   1:  PR[91,1] = PR[90,1] + -34.385;
   1:  PR[91,2] = PR[90,2] + -12.687;
   1:L PR[91] R[100]mm/sec CNT100;
   1:  PR[91,1] = PR[90,1] + -33.183;
   1:  PR[91,2] = PR[90,2] + -13.979;
   1:L PR[91] R[100]mm/sec CNT100;
   1:  PR[91,1] = PR[90,1] + -31.805;
   1:  PR[91,2] = PR[90,2] + -15.148;
   1:L PR[91] R[100]mm/sec CNT100;
   1:  PR[91,1] = PR[90,1] + -30.132;
   1:  PR[91,2] = PR[90,2] + -16.456;
   1:L PR[91] R[100]mm/sec CNT100;
   1:  PR[91,1] = PR[90,1] + -27.677;
   1:  PR[91,2] = PR[90,2] + -17.817;
   1:L PR[91] R[100]mm/sec CNT100;
   1:  PR[91,1] = PR[90,1] + -27.017;
   1:  PR[91,2] = PR[90,2] + -18.151;
   1:L PR[91] R[100]mm/sec CNT100;
   1:  PR[91,1] = PR[90,1] + -24.103;
   1:  PR[91,2] = PR[90,2] + -19.209;
   1:L PR[91] R[100]mm/sec CNT100;
   1:  PR[91,1] = PR[90,1] + -20.848;
   1:  PR[91,2] = PR[90,2] + -19.885;
   1:L PR[91] R[100]mm/sec CNT100;
   1:  PR[91,1] = PR[90,1] + -20.625;
   1:  PR[91,2] = PR[90,2] + -19.911;
   1:L PR[91] R[100]mm/sec CNT100;
   1:  PR[91,1] = PR[90,1] + -17.368;
   1:  PR[91,2] = PR[90,2] + -20.082;
   1:L PR[91] R[100]mm/sec CNT100;
   1:  PR[91,1] = PR[90,1] + -14.474;
   1:  PR[91,2] = PR[90,2] + -19.791;
   1:L PR[91] R[100]mm/sec CNT100;
   1:  PR[91,1] = PR[90,1] + -13.607;
   1:  PR[91,2] = PR[90,2] + -19.670;
   1:L PR[91] R[100]mm/sec CNT100;
   1:  PR[91,1] = PR[90,1] + -10.936;
   1:  PR[91,2] = PR[90,2] + -18.979;
   1:L PR[91] R[100]mm/sec CNT100;
   1:  PR[91,1] = PR[90,1] + -8.588;
   1:  PR[91,2] = PR[90,2] + -17.949;
   1:L PR[91] R[100]mm/sec CNT100;
   1:  PR[91,1] = PR[90,1] + -7.248;
   1:  PR[91,2] = PR[90,2] + -17.378;
   1:L PR[91] R[100]mm/sec CNT100;
   1:  PR[91,1] = PR[90,1] + -5.237;
   1:  PR[91,2] = PR[90,2] + -16.092;
   1:L PR[91] R[100]mm/sec CNT100;
   1:  PR[91,1] = PR[90,1] + -4.843;
   1:  PR[91,2] = PR[90,2] + -15.808;
   1:L PR[91] R[100]mm/sec CNT100;
   1:  PR[91,1] = PR[90,1] + -2.769;
   1:  PR[91,2] = PR[90,2] + -13.975;
   1:L PR[91] R[100]mm/sec CNT100;
   1:  PR[91,1] = PR[90,1] + -2.120;
   1:  PR[91,2] = PR[90,2] + -13.214;
   1:L PR[91] R[100]mm/sec CNT100;
   1:  PR[91,1] = PR[90,1] + -1.676;
   1:  PR[91,2] = PR[90,2] + -12.857;
   1:L PR[91] R[100]mm/sec CNT100;
   1:  PR[91,1] = PR[90,1] + -0.501;
   1:  PR[91,2] = PR[90,2] + -12.027;
   1:L PR[91] R[100]mm/sec CNT100;
   1:  PR[91,1] = PR[90,1] + 0.440;
   1:  PR[91,2] = PR[90,2] + -12.361;
   1:L PR[91] R[100]mm/sec CNT100;
   1:  PR[91,1] = PR[90,1] + 1.193;
   1:L PR[91] R[100]mm/sec CNT100;
   1:  PR[91,1] = PR[90,1] + 1.817;
   1:  PR[91,2] = PR[90,2] + -12.872;
   1:L PR[91] R[100]mm/sec CNT100;
   1:  PR[91,1] = PR[90,1] + 2.256;
   1:  PR[91,2] = PR[90,2] + -13.184;
   1:L PR[91] R[100]mm/sec CNT100;
   1:  PR[91,1] = PR[90,1] + 2.936;
   1:  PR[91,2] = PR[90,2] + -13.984;
   1:L PR[91] R[100]mm/sec CNT100;
   1:  PR[91,1] = PR[90,1] + 4.982;
   1:  PR[91,2] = PR[90,2] + -15.795;
   1:L PR[91] R[100]mm/sec CNT100;
   1:  PR[91,1] = PR[90,1] + 6.799;
   1:  PR[91,2] = PR[90,2] + -16.959;
   1:L PR[91] R[100]mm/sec CNT100;
   1:  PR[91,1] = PR[90,1] + 7.427;
   1:  PR[91,2] = PR[90,2] + -17.391;
   1:L PR[91] R[100]mm/sec CNT100;
   1:  PR[91,1] = PR[90,1] + 11.082;
   1:  PR[91,2] = PR[90,2] + -18.974;
   1:L PR[91] R[100]mm/sec CNT100;
   1:  PR[91,1] = PR[90,1] + 13.736;
   1:  PR[91,2] = PR[90,2] + -19.662;
   1:L PR[91] R[100]mm/sec CNT100;
   1:  PR[91,1] = PR[90,1] + 16.945;
   1:  PR[91,2] = PR[90,2] + -19.998;
   1:L PR[91] R[100]mm/sec CNT100;
   1:  PR[91,1] = PR[90,1] + 17.542;
   1:  PR[91,2] = PR[90,2] + -20.081;
   1:L PR[91] R[100]mm/sec CNT100;
   1:  PR[91,1] = PR[90,1] + 20.757;
   1:  PR[91,2] = PR[90,2] + -19.914;
   1:L PR[91] R[100]mm/sec CNT100;
   1:  PR[91,1] = PR[90,1] + 20.981;
   1:  PR[91,2] = PR[90,2] + -19.888;
   1:L PR[91] R[100]mm/sec CNT100;
   1:  PR[91,1] = PR[90,1] + 24.231;
   1:  PR[91,2] = PR[90,2] + -19.216;
   1:L PR[91] R[100]mm/sec CNT100;
   1:  PR[91,1] = PR[90,1] + 27.158;
   1:  PR[91,2] = PR[90,2] + -18.158;
   1:L PR[91] R[100]mm/sec CNT100;
   1:  PR[91,1] = PR[90,1] + 27.815;
   1:  PR[91,2] = PR[90,2] + -17.826;
   1:L PR[91] R[100]mm/sec CNT100;
   1:  PR[91,1] = PR[90,1] + 30.243;
   1:  PR[91,2] = PR[90,2] + -16.487;
   1:L PR[91] R[100]mm/sec CNT100;
   1:  PR[91,1] = PR[90,1] + 31.424;
   1:  PR[91,2] = PR[90,2] + -15.490;
   1:L PR[91] R[100]mm/sec CNT100;
   1:  PR[91,1] = PR[90,1] + 33.327;
   1:  PR[91,2] = PR[90,2] + -13.989;
   1:L PR[91] R[100]mm/sec CNT100;
   1:  PR[91,1] = PR[90,1] + 34.543;
   1:  PR[91,2] = PR[90,2] + -12.683;
   1:L PR[91] R[100]mm/sec CNT100;
   1:  PR[91,1] = PR[90,1] + 35.930;
   1:  PR[91,2] = PR[90,2] + -10.746;
   1:L PR[91] R[100]mm/sec CNT100;
   1:  PR[91,1] = PR[90,1] + 36.829;
   1:  PR[91,2] = PR[90,2] + -9.386;
   1:L PR[91] R[100]mm/sec CNT100;
   1:  PR[91,1] = PR[90,1] + 37.404;
   1:  PR[91,2] = PR[90,2] + -8.113;
   1:L PR[91] R[100]mm/sec CNT100;
   1:  PR[91,1] = PR[90,1] + 38.431;
   1:  PR[91,2] = PR[90,2] + -5.567;
   1:L PR[91] R[100]mm/sec CNT100;
   1:  PR[91,1] = PR[90,1] + 38.718;
   1:  PR[91,2] = PR[90,2] + -4.469;
   1:L PR[91] R[100]mm/sec CNT100;
   1:  PR[91,1] = PR[90,1] + 39.102;
   1:  PR[91,2] = PR[90,2] + -1.437;
   1:L PR[91] R[100]mm/sec CNT100;
   1:  PR[91,1] = PR[90,1] + 39.190;
   1:  PR[91,2] = PR[90,2] + -0.345;
   1:L PR[91] R[100]mm/sec CNT100;
   1:  PR[91,1] = PR[90,1] + 38.810;
   1:  PR[91,2] = PR[90,2] + 2.635;
   1:L PR[91] R[100]mm/sec CNT100;
   1:  PR[91,1] = PR[90,1] + 38.710;
   1:  PR[91,2] = PR[90,2] + 3.878;
   1:L PR[91] R[100]mm/sec CNT100;
   1:  PR[91,1] = PR[90,1] + 38.430;
   1:  PR[91,2] = PR[90,2] + 4.944;
   1:L PR[91] R[100]mm/sec CNT100;
   1:  PR[91,1] = PR[90,1] + 37.403;
   1:  PR[91,2] = PR[90,2] + 7.490;
   1:L PR[91] R[100]mm/sec CNT100;
   1:  PR[91,1] = PR[90,1] + 36.840;
   1:  PR[91,2] = PR[90,2] + 8.736;
   1:L PR[91] R[100]mm/sec CNT100;
   1:  PR[91,1] = PR[90,1] + 35.420;
   1:  PR[91,2] = PR[90,2] + 10.708;
   1:L PR[91] R[100]mm/sec CNT100;
   1:  PR[91,1] = PR[90,1] + 34.521;
   1:  PR[91,2] = PR[90,2] + 12.083;
   1:L PR[91] R[100]mm/sec CNT100;
   1:  PR[91,1] = PR[90,1] + 33.307;
   1:  PR[91,2] = PR[90,2] + 13.386;
   1:L PR[91] R[100]mm/sec CNT100;
   1:  PR[91,1] = PR[90,1] + 31.932;
   1:  PR[91,2] = PR[90,2] + 14.555;
   1:L PR[91] R[100]mm/sec CNT100;
   1:  PR[91,1] = PR[90,1] + 30.267;
   1:  PR[91,2] = PR[90,2] + 15.850;
   1:L PR[91] R[100]mm/sec CNT100;
   1:  PR[91,1] = PR[90,1] + 27.814;
   1:  PR[91,2] = PR[90,2] + 17.202;
   1:L PR[91] R[100]mm/sec CNT100;
   1:  PR[91,1] = PR[90,1] + 27.157;
   1:  PR[91,2] = PR[90,2] + 17.534;
   1:L PR[91] R[100]mm/sec CNT100;
   1:  PR[91,1] = PR[90,1] + 24.231;
   1:  PR[91,2] = PR[90,2] + 18.592;
   1:L PR[91] R[100]mm/sec CNT100;
   1:  PR[91,1] = PR[90,1] + 20.982;
   1:  PR[91,2] = PR[90,2] + 19.264;
   1:L PR[91] R[100]mm/sec CNT100;
   1:  PR[91,1] = PR[90,1] + 20.758;
   1:  PR[91,2] = PR[90,2] + 19.290;
   1:L PR[91] R[100]mm/sec CNT100;
   1:  PR[91,1] = PR[90,1] + 17.520;
   1:  PR[91,2] = PR[90,2] + 19.459;
   1:L PR[91] R[100]mm/sec CNT100;
   1:  PR[91,1] = PR[90,1] + 14.634;
   1:  PR[91,2] = PR[90,2] + 19.166;
   1:L PR[91] R[100]mm/sec CNT100;
   1:  PR[91,1] = PR[90,1] + 13.768;
   1:  PR[91,2] = PR[90,2] + 19.046;
   1:L PR[91] R[100]mm/sec CNT100;
   1:  PR[91,1] = PR[90,1] + 11.095;
   1:  PR[91,2] = PR[90,2] + 18.353;
   1:L PR[91] R[100]mm/sec CNT100;
   1:  PR[91,1] = PR[90,1] + 8.749;
   1:  PR[91,2] = PR[90,2] + 17.327;
   1:L PR[91] R[100]mm/sec CNT100;
   1:  PR[91,1] = PR[90,1] + 7.438;
   1:  PR[91,2] = PR[90,2] + 16.779;
   1:L PR[91] R[100]mm/sec CNT100;
   1:  PR[91,1] = PR[90,1] + 5.424;
   1:  PR[91,2] = PR[90,2] + 15.493;
   1:L PR[91] R[100]mm/sec CNT100;
   1:  PR[91,1] = PR[90,1] + 5.171;
   1:  PR[91,2] = PR[90,2] + 15.318;
   1:L PR[91] R[100]mm/sec CNT100;
   1:  PR[91,1] = PR[90,1] + 4.692;
   1:  PR[91,2] = PR[90,2] + 14.939;
   1:L PR[91] R[100]mm/sec CNT100;
   1:  PR[91,1] = PR[90,1] + 3.034;
   1:  PR[91,2] = PR[90,2] + 13.458;
   1:L PR[91] R[100]mm/sec CNT100;
   1:  PR[91,1] = PR[90,1] + 2.330;
   1:  PR[91,2] = PR[90,2] + 12.730;
   1:L PR[91] R[100]mm/sec CNT100;
   1:  PR[91,1] = PR[90,1] + 2.090;
   1:  PR[91,2] = PR[90,2] + 12.413;
   1:L PR[91] R[100]mm/sec CNT100;
   1:  PR[91,1] = PR[90,1] + 1.443;
   1:  PR[91,2] = PR[90,2] + 11.955;
   1:L PR[91] R[100]mm/sec CNT100;
   1:  PR[91,1] = PR[90,1] + 0.740;
   1:  PR[91,2] = PR[90,2] + 11.570;
   1:L PR[91] R[100]mm/sec CNT100;
   1:  PR[91,1] = PR[90,1] + -0.586;
   1:L PR[91] R[100]mm/sec CNT100;
   1:  PR[91] = PR[90];
   1:  PR[91,1] = PR[90,1] + -1.541;
   1:  PR[91,2] = PR[90,2] + 12.321;
   1:  PR[91,3] = PR[90,3] + 28.365;
   1:L PR[91] R[100]mm/sec CNT100;
   1:  PR[91,1] = PR[90,1] + -1.870;
   1:  PR[91,2] = PR[90,2] + 12.749;
   1:L PR[91] R[100]mm/sec CNT100;
   1:  PR[91,1] = PR[90,1] + -2.109;
   1:  PR[91,2] = PR[90,2] + 12.974;
   1:L PR[91] R[100]mm/sec CNT100;
   1:  PR[91,1] = PR[90,1] + -2.678;
   1:  PR[91,2] = PR[90,2] + 13.569;
   1:L PR[91] R[100]mm/sec CNT100;
   1:  PR[91,1] = PR[90,1] + -4.236;
   1:  PR[91,2] = PR[90,2] + 14.958;
   1:L PR[91] R[100]mm/sec CNT100;
   1:  PR[91,1] = PR[90,1] + -4.761;
   1:  PR[91,2] = PR[90,2] + 15.373;
   1:L PR[91] R[100]mm/sec CNT100;
   1:  PR[91,1] = PR[90,1] + -6.588;
   1:  PR[91,2] = PR[90,2] + 16.543;
   1:L PR[91] R[100]mm/sec CNT100;
   1:  PR[91,1] = PR[90,1] + -7.022;
   1:  PR[91,2] = PR[90,2] + 16.834;
   1:L PR[91] R[100]mm/sec CNT100;
   1:  PR[91,1] = PR[90,1] + -9.377;
   1:  PR[91,2] = PR[90,2] + 17.863;
   1:L PR[91] R[100]mm/sec CNT100;
   1:  PR[91,1] = PR[90,1] + -10.739;
   1:  PR[91,2] = PR[90,2] + 18.434;
   1:L PR[91] R[100]mm/sec CNT100;
   1:  PR[91,1] = PR[90,1] + -13.266;
   1:  PR[91,2] = PR[90,2] + 19.087;
   1:L PR[91] R[100]mm/sec CNT100;
   1:  PR[91,1] = PR[90,1] + -16.330;
   1:  PR[91,2] = PR[90,2] + 19.406;
   1:L PR[91] R[100]mm/sec CNT100;
   1:  PR[91,1] = PR[90,1] + -17.174;
   1:  PR[91,2] = PR[90,2] + 19.521;
   1:L PR[91] R[100]mm/sec CNT100;
   1:  PR[91,1] = PR[90,1] + -20.260;
   1:  PR[91,2] = PR[90,2] + 19.358;
   1:L PR[91] R[100]mm/sec CNT100;
   1:  PR[91,1] = PR[90,1] + -20.724;
   1:  PR[91,2] = PR[90,2] + 19.304;
   1:L PR[91] R[100]mm/sec CNT100;
   1:  PR[91,1] = PR[90,1] + -23.832;
   1:  PR[91,2] = PR[90,2] + 18.659;
   1:L PR[91] R[100]mm/sec CNT100;
   1:  PR[91,1] = PR[90,1] + -26.964;
   1:  PR[91,2] = PR[90,2] + 17.504;
   1:L PR[91] R[100]mm/sec CNT100;
   1:  PR[91,1] = PR[90,1] + -29.926;
   1:  PR[91,2] = PR[90,2] + 15.872;
   1:L PR[91] R[100]mm/sec CNT100;
   1:  PR[91,1] = PR[90,1] + -30.643;
   1:  PR[91,2] = PR[90,2] + 15.268;
   1:L PR[91] R[100]mm/sec CNT100;
   1:  PR[91,1] = PR[90,1] + -32.892;
   1:  PR[91,2] = PR[90,2] + 13.488;
   1:L PR[91] R[100]mm/sec CNT100;
   1:  PR[91,1] = PR[90,1] + -34.331;
   1:  PR[91,2] = PR[90,2] + 11.939;
   1:L PR[91] R[100]mm/sec CNT100;
   1:  PR[91,1] = PR[90,1] + -35.417;
   1:  PR[91,2] = PR[90,2] + 10.423;
   1:L PR[91] R[100]mm/sec CNT100;
   1:  PR[91,1] = PR[90,1] + -36.499;
   1:  PR[91,2] = PR[90,2] + 8.777;
   1:L PR[91] R[100]mm/sec CNT100;
   1:  PR[91,1] = PR[90,1] + -37.206;
   1:  PR[91,2] = PR[90,2] + 7.190;
   1:L PR[91] R[100]mm/sec CNT100;
   1:  PR[91,1] = PR[90,1] + -38.062;
   1:  PR[91,2] = PR[90,2] + 5.058;
   1:L PR[91] R[100]mm/sec CNT100;
   1:  PR[91,1] = PR[90,1] + -38.428;
   1:  PR[91,2] = PR[90,2] + 3.643;
   1:L PR[91] R[100]mm/sec CNT100;
   1:  PR[91,1] = PR[90,1] + -38.751;
   1:  PR[91,2] = PR[90,2] + 1.099;
   1:L PR[91] R[100]mm/sec CNT100;
   1:  PR[91,1] = PR[90,1] + -38.860;
   1:  PR[91,2] = PR[90,2] + -0.277;
   1:L PR[91] R[100]mm/sec CNT100;
   1:  PR[91,1] = PR[90,1] + -38.538;
   1:  PR[91,2] = PR[90,2] + -2.788;
   1:L PR[91] R[100]mm/sec CNT100;
   1:  PR[91,1] = PR[90,1] + -38.420;
   1:  PR[91,2] = PR[90,2] + -4.301;
   1:L PR[91] R[100]mm/sec CNT100;
   1:  PR[91,1] = PR[90,1] + -38.062;
   1:  PR[91,2] = PR[90,2] + -5.682;
   1:L PR[91] R[100]mm/sec CNT100;
   1:  PR[91,1] = PR[90,1] + -37.206;
   1:  PR[91,2] = PR[90,2] + -7.814;
   1:L PR[91] R[100]mm/sec CNT100;
   1:  PR[91,1] = PR[90,1] + -36.512;
   1:  PR[91,2] = PR[90,2] + -9.372;
   1:L PR[91] R[100]mm/sec CNT100;
   1:  PR[91,1] = PR[90,1] + -35.356;
   1:  PR[91,2] = PR[90,2] + -10.976;
   1:L PR[91] R[100]mm/sec CNT100;
   1:  PR[91,1] = PR[90,1] + -34.309;
   1:  PR[91,2] = PR[90,2] + -12.587;
   1:L PR[91] R[100]mm/sec CNT100;
   1:  PR[91,1] = PR[90,1] + -32.875;
   1:  PR[91,2] = PR[90,2] + -14.130;
   1:L PR[91] R[100]mm/sec CNT100;
   1:  PR[91,1] = PR[90,1] + -31.875;
   1:  PR[91,2] = PR[90,2] + -14.979;
   1:L PR[91] R[100]mm/sec CNT100;
   1:  PR[91,1] = PR[90,1] + -29.950;
   1:  PR[91,2] = PR[90,2] + -16.483;
   1:L PR[91] R[100]mm/sec CNT100;
   1:  PR[91,1] = PR[90,1] + -26.964;
   1:  PR[91,2] = PR[90,2] + -18.128;
   1:L PR[91] R[100]mm/sec CNT100;
   1:  PR[91,1] = PR[90,1] + -23.830;
   1:  PR[91,2] = PR[90,2] + -19.283;
   1:L PR[91] R[100]mm/sec CNT100;
   1:  PR[91,1] = PR[90,1] + -20.722;
   1:  PR[91,2] = PR[90,2] + -19.928;
   1:L PR[91] R[100]mm/sec CNT100;
   1:  PR[91,1] = PR[90,1] + -20.256;
   1:  PR[91,2] = PR[90,2] + -19.982;
   1:L PR[91] R[100]mm/sec CNT100;
   1:  PR[91,1] = PR[90,1] + -17.142;
   1:  PR[91,2] = PR[90,2] + -20.146;
   1:L PR[91] R[100]mm/sec CNT100;
   1:  PR[91,1] = PR[90,1] + -14.376;
   1:  PR[91,2] = PR[90,2] + -19.868;
   1:L PR[91] R[100]mm/sec CNT100;
   1:  PR[91,1] = PR[90,1] + -13.279;
   1:  PR[91,2] = PR[90,2] + -19.714;
   1:L PR[91] R[100]mm/sec CNT100;
   1:  PR[91,1] = PR[90,1] + -10.738;
   1:  PR[91,2] = PR[90,2] + -19.057;
   1:L PR[91] R[100]mm/sec CNT100;
   1:  PR[91,1] = PR[90,1] + -8.500;
   1:  PR[91,2] = PR[90,2] + -18.076;
   1:L PR[91] R[100]mm/sec CNT100;
   1:  PR[91,1] = PR[90,1] + -6.954;
   1:  PR[91,2] = PR[90,2] + -17.417;
   1:L PR[91] R[100]mm/sec CNT100;
   1:  PR[91,1] = PR[90,1] + -5.052;
   1:  PR[91,2] = PR[90,2] + -16.201;
   1:L PR[91] R[100]mm/sec CNT100;
   1:  PR[91,1] = PR[90,1] + -4.596;
   1:  PR[91,2] = PR[90,2] + -15.871;
   1:L PR[91] R[100]mm/sec CNT100;
   1:  PR[91,1] = PR[90,1] + -2.999;
   1:  PR[91,2] = PR[90,2] + -14.474;
   1:L PR[91] R[100]mm/sec CNT100;
   1:  PR[91,1] = PR[90,1] + -2.567;
   1:  PR[91,2] = PR[90,2] + -14.085;
   1:L PR[91] R[100]mm/sec CNT100;
   1:  PR[91,1] = PR[90,1] + -2.101;
   1:  PR[91,2] = PR[90,2] + -13.539;
   1:L PR[91] R[100]mm/sec CNT100;
   1:  PR[91,1] = PR[90,1] + -1.599;
   1:  PR[91,2] = PR[90,2] + -13.135;
   1:L PR[91] R[100]mm/sec CNT100;
   1:  PR[91,1] = PR[90,1] + -0.477;
   1:  PR[91,2] = PR[90,2] + -12.341;
   1:L PR[91] R[100]mm/sec CNT100;
   1:  PR[91,1] = PR[90,1] + 0.564;
   1:  PR[91,2] = PR[90,2] + -12.711;
   1:L PR[91] R[100]mm/sec CNT100;
   1:  PR[91,1] = PR[90,1] + 1.217;
   1:L PR[91] R[100]mm/sec CNT100;
   1:  PR[91,1] = PR[90,1] + 1.898;
   1:  PR[91,2] = PR[90,2] + -13.268;
   1:L PR[91] R[100]mm/sec CNT100;
   1:  PR[91,1] = PR[90,1] + 2.236;
   1:  PR[91,2] = PR[90,2] + -13.509;
   1:L PR[91] R[100]mm/sec CNT100;
   1:  PR[91,1] = PR[90,1] + 2.727;
   1:  PR[91,2] = PR[90,2] + -14.086;
   1:L PR[91] R[100]mm/sec CNT100;
   1:  PR[91,1] = PR[90,1] + 4.736;
   1:  PR[91,2] = PR[90,2] + -15.859;
   1:L PR[91] R[100]mm/sec CNT100;
   1:  PR[91,1] = PR[90,1] + 6.403;
   1:  PR[91,2] = PR[90,2] + -16.926;
   1:L PR[91] R[100]mm/sec CNT100;
   1:  PR[91,1] = PR[90,1] + 7.134;
   1:  PR[91,2] = PR[90,2] + -17.430;
   1:L PR[91] R[100]mm/sec CNT100;
   1:  PR[91,1] = PR[90,1] + 10.884;
   1:  PR[91,2] = PR[90,2] + -19.052;
   1:L PR[91] R[100]mm/sec CNT100;
   1:  PR[91,1] = PR[90,1] + 13.409;
   1:  PR[91,2] = PR[90,2] + -19.707;
   1:L PR[91] R[100]mm/sec CNT100;
   1:  PR[91,1] = PR[90,1] + 16.470;
   1:  PR[91,2] = PR[90,2] + -20.028;
   1:L PR[91] R[100]mm/sec CNT100;
   1:  PR[91,1] = PR[90,1] + 17.317;
   1:  PR[91,2] = PR[90,2] + -20.145;
   1:L PR[91] R[100]mm/sec CNT100;
   1:  PR[91,1] = PR[90,1] + 20.388;
   1:  PR[91,2] = PR[90,2] + -19.986;
   1:L PR[91] R[100]mm/sec CNT100;
   1:  PR[91,1] = PR[90,1] + 20.856;
   1:  PR[91,2] = PR[90,2] + -19.931;
   1:L PR[91] R[100]mm/sec CNT100;
   1:  PR[91,1] = PR[90,1] + 23.960;
   1:  PR[91,2] = PR[90,2] + -19.289;
   1:L PR[91] R[100]mm/sec CNT100;
   1:  PR[91,1] = PR[90,1] + 27.104;
   1:  PR[91,2] = PR[90,2] + -18.135;
   1:L PR[91] R[100]mm/sec CNT100;
   1:  PR[91,1] = PR[90,1] + 30.057;
   1:  PR[91,2] = PR[90,2] + -16.516;
   1:L PR[91] R[100]mm/sec CNT100;
   1:  PR[91,1] = PR[90,1] + 30.770;
   1:  PR[91,2] = PR[90,2] + -15.915;
   1:L PR[91] R[100]mm/sec CNT100;
   1:  PR[91,1] = PR[90,1] + 33.013;
   1:  PR[91,2] = PR[90,2] + -14.145;
   1:L PR[91] R[100]mm/sec CNT100;
   1:  PR[91,1] = PR[90,1] + 34.463;
   1:  PR[91,2] = PR[90,2] + -12.587;
   1:L PR[91] R[100]mm/sec CNT100;
   1:  PR[91,1] = PR[90,1] + 35.549;
   1:  PR[91,2] = PR[90,2] + -11.071;
   1:L PR[91] R[100]mm/sec CNT100;
   1:  PR[91,1] = PR[90,1] + 36.650;
   1:  PR[91,2] = PR[90,2] + -9.405;
   1:L PR[91] R[100]mm/sec CNT100;
   1:  PR[91,1] = PR[90,1] + 37.356;
   1:  PR[91,2] = PR[90,2] + -7.841;
   1:L PR[91] R[100]mm/sec CNT100;
   1:  PR[91,1] = PR[90,1] + 38.211;
   1:  PR[91,2] = PR[90,2] + -5.722;
   1:L PR[91] R[100]mm/sec CNT100;
   1:  PR[91,1] = PR[90,1] + 38.578;
   1:  PR[91,2] = PR[90,2] + -4.323;
   1:L PR[91] R[100]mm/sec CNT100;
   1:  PR[91,1] = PR[90,1] + 38.901;
   1:  PR[91,2] = PR[90,2] + -1.769;
   1:L PR[91] R[100]mm/sec CNT100;
   1:  PR[91,1] = PR[90,1] + 39.016;
   1:  PR[91,2] = PR[90,2] + -0.345;
   1:L PR[91] R[100]mm/sec CNT100;
   1:  PR[91,1] = PR[90,1] + 38.695;
   1:  PR[91,2] = PR[90,2] + 2.173;
   1:L PR[91] R[100]mm/sec CNT100;
   1:  PR[91,1] = PR[90,1] + 38.570;
   1:  PR[91,2] = PR[90,2] + 3.732;
   1:L PR[91] R[100]mm/sec CNT100;
   1:  PR[91,1] = PR[90,1] + 38.211;
   1:  PR[91,2] = PR[90,2] + 5.098;
   1:L PR[91] R[100]mm/sec CNT100;
   1:  PR[91,1] = PR[90,1] + 37.355;
   1:  PR[91,2] = PR[90,2] + 7.219;
   1:L PR[91] R[100]mm/sec CNT100;
   1:  PR[91,1] = PR[90,1] + 36.661;
   1:  PR[91,2] = PR[90,2] + 8.756;
   1:L PR[91] R[100]mm/sec CNT100;
   1:  PR[91,1] = PR[90,1] + 35.505;
   1:  PR[91,2] = PR[90,2] + 10.362;
   1:L PR[91] R[100]mm/sec CNT100;
   1:  PR[91,1] = PR[90,1] + 34.441;
   1:  PR[91,2] = PR[90,2] + 11.987;
   1:L PR[91] R[100]mm/sec CNT100;
   1:  PR[91,1] = PR[90,1] + 32.994;
   1:  PR[91,2] = PR[90,2] + 13.541;
   1:L PR[91] R[100]mm/sec CNT100;
   1:  PR[91,1] = PR[90,1] + 31.998;
   1:  PR[91,2] = PR[90,2] + 14.388;
   1:L PR[91] R[100]mm/sec CNT100;
   1:  PR[91,1] = PR[90,1] + 30.082;
   1:  PR[91,2] = PR[90,2] + 15.879;
   1:L PR[91] R[100]mm/sec CNT100;
   1:  PR[91,1] = PR[90,1] + 27.103;
   1:  PR[91,2] = PR[90,2] + 17.511;
   1:L PR[91] R[100]mm/sec CNT100;
   1:  PR[91,1] = PR[90,1] + 23.962;
   1:  PR[91,2] = PR[90,2] + 18.664;
   1:L PR[91] R[100]mm/sec CNT100;
   1:  PR[91,1] = PR[90,1] + 20.858;
   1:  PR[91,2] = PR[90,2] + 19.307;
   1:L PR[91] R[100]mm/sec CNT100;
   1:  PR[91,1] = PR[90,1] + 20.392;
   1:  PR[91,2] = PR[90,2] + 19.362;
   1:L PR[91] R[100]mm/sec CNT100;
   1:  PR[91,1] = PR[90,1] + 17.296;
   1:  PR[91,2] = PR[90,2] + 19.523;
   1:L PR[91] R[100]mm/sec CNT100;
   1:  PR[91,1] = PR[90,1] + 14.537;
   1:  PR[91,2] = PR[90,2] + 19.243;
   1:L PR[91] R[100]mm/sec CNT100;
   1:  PR[91,1] = PR[90,1] + 13.443;
   1:  PR[91,2] = PR[90,2] + 19.092;
   1:L PR[91] R[100]mm/sec CNT100;
   1:  PR[91,1] = PR[90,1] + 10.900;
   1:  PR[91,2] = PR[90,2] + 18.432;
   1:L PR[91] R[100]mm/sec CNT100;
   1:  PR[91,1] = PR[90,1] + 8.663;
   1:  PR[91,2] = PR[90,2] + 17.454;
   1:L PR[91] R[100]mm/sec CNT100;
   1:  PR[91,1] = PR[90,1] + 7.150;
   1:  PR[91,2] = PR[90,2] + 16.822;
   1:L PR[91] R[100]mm/sec CNT100;
   1:  PR[91,1] = PR[90,1] + 5.242;
   1:  PR[91,2] = PR[90,2] + 15.603;
   1:L PR[91] R[100]mm/sec CNT100;
   1:  PR[91,1] = PR[90,1] + 4.950;
   1:  PR[91,2] = PR[90,2] + 15.401;
   1:L PR[91] R[100]mm/sec CNT100;
   1:  PR[91,1] = PR[90,1] + 4.403;
   1:  PR[91,2] = PR[90,2] + 14.969;
   1:L PR[91] R[100]mm/sec CNT100;
   1:  PR[91,1] = PR[90,1] + 2.844;
   1:  PR[91,2] = PR[90,2] + 13.578;
   1:L PR[91] R[100]mm/sec CNT100;
   1:  PR[91,1] = PR[90,1] + 2.206;
   1:  PR[91,2] = PR[90,2] + 12.907;
   1:L PR[91] R[100]mm/sec CNT100;
   1:  PR[91,1] = PR[90,1] + 2.161;
   1:  PR[91,2] = PR[90,2] + 12.875;
   1:L PR[91] R[100]mm/sec CNT100;
   1:  PR[91,1] = PR[90,1] + 2.032;
   1:  PR[91,2] = PR[90,2] + 12.705;
   1:L PR[91] R[100]mm/sec CNT100;
   1:  PR[91,1] = PR[90,1] + 1.467;
   1:  PR[91,2] = PR[90,2] + 12.305;
   1:L PR[91] R[100]mm/sec CNT100;
   1:  PR[91,1] = PR[90,1] + 0.699;
   1:  PR[91,2] = PR[90,2] + 11.885;
   1:L PR[91] R[100]mm/sec CNT100;
   1:  PR[91,1] = PR[90,1] + -0.562;
   1:  PR[91,2] = PR[90,2] + 11.884;
   1:L PR[91] R[100]mm/sec CNT100;
   1:  PR[91] = PR[90];
   1:  PR[91,1] = PR[90,1] + -1.580;
   1:  PR[91,2] = PR[90,2] + 12.664;
   1:  PR[91,3] = PR[90,3] + 28.975;
   1:L PR[91] R[100]mm/sec CNT100;
   1:  PR[91,1] = PR[90,1] + -1.940;
   1:  PR[91,2] = PR[90,2] + 13.132;
   1:L PR[91] R[100]mm/sec CNT100;
   1:  PR[91,1] = PR[90,1] + -2.091;
   1:  PR[91,2] = PR[90,2] + 13.274;
   1:L PR[91] R[100]mm/sec CNT100;
   1:  PR[91,1] = PR[90,1] + -2.485;
   1:  PR[91,2] = PR[90,2] + 13.687;
   1:L PR[91] R[100]mm/sec CNT100;
   1:  PR[91,1] = PR[90,1] + -3.950;
   1:  PR[91,2] = PR[90,2] + 14.989;
   1:L PR[91] R[100]mm/sec CNT100;
   1:  PR[91,1] = PR[90,1] + -4.541;
   1:  PR[91,2] = PR[90,2] + 15.457;
   1:L PR[91] R[100]mm/sec CNT100;
   1:  PR[91,1] = PR[90,1] + -6.235;
   1:  PR[91,2] = PR[90,2] + 16.541;
   1:L PR[91] R[100]mm/sec CNT100;
   1:  PR[91,1] = PR[90,1] + -6.735;
   1:  PR[91,2] = PR[90,2] + 16.877;
   1:L PR[91] R[100]mm/sec CNT100;
   1:  PR[91,1] = PR[90,1] + -8.963;
   1:  PR[91,2] = PR[90,2] + 17.850;
   1:L PR[91] R[100]mm/sec CNT100;
   1:  PR[91,1] = PR[90,1] + -10.543;
   1:  PR[91,2] = PR[90,2] + 18.513;
   1:L PR[91] R[100]mm/sec CNT100;
   1:  PR[91,1] = PR[90,1] + -12.941;
   1:  PR[91,2] = PR[90,2] + 19.133;
   1:L PR[91] R[100]mm/sec CNT100;
   1:  PR[91,1] = PR[90,1] + -15.857;
   1:  PR[91,2] = PR[90,2] + 19.436;
   1:L PR[91] R[100]mm/sec CNT100;
   1:  PR[91,1] = PR[90,1] + -16.950;
   1:  PR[91,2] = PR[90,2] + 19.585;
   1:L PR[91] R[100]mm/sec CNT100;
   1:  PR[91,1] = PR[90,1] + -19.892;
   1:  PR[91,2] = PR[90,2] + 19.430;
   1:L PR[91] R[100]mm/sec CNT100;
   1:  PR[91,1] = PR[90,1] + -20.599;
   1:  PR[91,2] = PR[90,2] + 19.346;
   1:L PR[91] R[100]mm/sec CNT100;
   1:  PR[91,1] = PR[90,1] + -23.571;
   1:  PR[91,2] = PR[90,2] + 18.730;
   1:L PR[91] R[100]mm/sec CNT100;
   1:  PR[91,1] = PR[90,1] + -26.859;
   1:  PR[91,2] = PR[90,2] + 17.507;
   1:L PR[91] R[100]mm/sec CNT100;
   1:  PR[91,1] = PR[90,1] + -29.739;
   1:  PR[91,2] = PR[90,2] + 15.903;
   1:L PR[91] R[100]mm/sec CNT100;
   1:  PR[91,1] = PR[90,1] + -29.993;
   1:  PR[91,2] = PR[90,2] + 15.689;
   1:L PR[91] R[100]mm/sec CNT100;
   1:  PR[91,1] = PR[90,1] + -32.584;
   1:  PR[91,2] = PR[90,2] + 13.638;
   1:L PR[91] R[100]mm/sec CNT100;
   1:  PR[91,1] = PR[90,1] + -34.255;
   1:  PR[91,2] = PR[90,2] + 11.840;
   1:L PR[91] R[100]mm/sec CNT100;
   1:  PR[91,1] = PR[90,1] + -35.041;
   1:  PR[91,2] = PR[90,2] + 10.743;
   1:L PR[91] R[100]mm/sec CNT100;
   1:  PR[91,1] = PR[90,1] + -36.322;
   1:  PR[91,2] = PR[90,2] + 8.794;
   1:L PR[91] R[100]mm/sec CNT100;
   1:  PR[91,1] = PR[90,1] + -37.160;
   1:  PR[91,2] = PR[90,2] + 6.913;
   1:L PR[91] R[100]mm/sec CNT100;
   1:  PR[91,1] = PR[90,1] + -37.845;
   1:  PR[91,2] = PR[90,2] + 5.208;
   1:L PR[91] R[100]mm/sec CNT100;
   1:  PR[91,1] = PR[90,1] + -38.289;
   1:  PR[91,2] = PR[90,2] + 3.489;
   1:L PR[91] R[100]mm/sec CNT100;
   1:  PR[91,1] = PR[90,1] + -38.551;
   1:  PR[91,2] = PR[90,2] + 1.422;
   1:L PR[91] R[100]mm/sec CNT100;
   1:  PR[91,1] = PR[90,1] + -38.686;
   1:  PR[91,2] = PR[90,2] + -0.277;
   1:L PR[91] R[100]mm/sec CNT100;
   1:  PR[91,1] = PR[90,1] + -38.423;
   1:  PR[91,2] = PR[90,2] + -2.328;
   1:L PR[91] R[100]mm/sec CNT100;
   1:  PR[91,1] = PR[90,1] + -38.280;
   1:  PR[91,2] = PR[90,2] + -4.147;
   1:L PR[91] R[100]mm/sec CNT100;
   1:  PR[91,1] = PR[90,1] + -37.845;
   1:  PR[91,2] = PR[90,2] + -5.832;
   1:L PR[91] R[100]mm/sec CNT100;
   1:  PR[91,1] = PR[90,1] + -37.160;
   1:  PR[91,2] = PR[90,2] + -7.537;
   1:L PR[91] R[100]mm/sec CNT100;
   1:  PR[91,1] = PR[90,1] + -36.335;
   1:  PR[91,2] = PR[90,2] + -9.389;
   1:L PR[91] R[100]mm/sec CNT100;
   1:  PR[91,1] = PR[90,1] + -35.442;
   1:  PR[91,2] = PR[90,2] + -10.629;
   1:L PR[91] R[100]mm/sec CNT100;
   1:  PR[91,1] = PR[90,1] + -34.233;
   1:  PR[91,2] = PR[90,2] + -12.488;
   1:L PR[91] R[100]mm/sec CNT100;
   1:  PR[91,1] = PR[90,1] + -32.567;
   1:  PR[91,2] = PR[90,2] + -14.280;
   1:L PR[91] R[100]mm/sec CNT100;
   1:  PR[91,1] = PR[90,1] + -31.944;
   1:  PR[91,2] = PR[90,2] + -14.809;
   1:L PR[91] R[100]mm/sec CNT100;
   1:  PR[91,1] = PR[90,1] + -29.763;
   1:  PR[91,2] = PR[90,2] + -16.514;
   1:L PR[91] R[100]mm/sec CNT100;
   1:  PR[91,1] = PR[90,1] + -26.858;
   1:  PR[91,2] = PR[90,2] + -18.131;
   1:L PR[91] R[100]mm/sec CNT100;
   1:  PR[91,1] = PR[90,1] + -23.568;
   1:  PR[91,2] = PR[90,2] + -19.354;
   1:L PR[91] R[100]mm/sec CNT100;
   1:  PR[91,1] = PR[90,1] + -20.595;
   1:  PR[91,2] = PR[90,2] + -19.971;
   1:L PR[91] R[100]mm/sec CNT100;
   1:  PR[91,1] = PR[90,1] + -19.887;
   1:  PR[91,2] = PR[90,2] + -20.054;
   1:L PR[91] R[100]mm/sec CNT100;
   1:  PR[91,1] = PR[90,1] + -16.916;
   1:  PR[91,2] = PR[90,2] + -20.211;
   1:L PR[91] R[100]mm/sec CNT100;
   1:  PR[91,1] = PR[90,1] + -14.277;
   1:  PR[91,2] = PR[90,2] + -19.945;
   1:L PR[91] R[100]mm/sec CNT100;
   1:  PR[91,1] = PR[90,1] + -12.953;
   1:  PR[91,2] = PR[90,2] + -19.759;
   1:L PR[91] R[100]mm/sec CNT100;
   1:  PR[91,1] = PR[90,1] + -10.540;
   1:  PR[91,2] = PR[90,2] + -19.136;
   1:L PR[91] R[100]mm/sec CNT100;
   1:  PR[91,1] = PR[90,1] + -8.413;
   1:  PR[91,2] = PR[90,2] + -18.203;
   1:L PR[91] R[100]mm/sec CNT100;
   1:  PR[91,1] = PR[90,1] + -6.661;
   1:  PR[91,2] = PR[90,2] + -17.456;
   1:L PR[91] R[100]mm/sec CNT100;
   1:  PR[91,1] = PR[90,1] + -4.867;
   1:  PR[91,2] = PR[90,2] + -16.309;
   1:L PR[91] R[100]mm/sec CNT100;
   1:  PR[91,1] = PR[90,1] + -4.353;
   1:  PR[91,2] = PR[90,2] + -15.938;
   1:L PR[91] R[100]mm/sec CNT100;
   1:  PR[91,1] = PR[90,1] + -2.355;
   1:  PR[91,2] = PR[90,2] + -14.182;
   1:L PR[91] R[100]mm/sec CNT100;
   1:  PR[91,1] = PR[90,1] + -2.083;
   1:  PR[91,2] = PR[90,2] + -13.863;
   1:L PR[91] R[100]mm/sec CNT100;
   1:  PR[91,1] = PR[90,1] + -1.522;
   1:  PR[91,2] = PR[90,2] + -13.413;
   1:L PR[91] R[100]mm/sec CNT100;
   1:  PR[91,1] = PR[90,1] + -0.452;
   1:  PR[91,2] = PR[90,2] + -12.656;
   1:L PR[91] R[100]mm/sec CNT100;
   1:  PR[91,1] = PR[90,1] + 0.687;
   1:  PR[91,2] = PR[90,2] + -13.061;
   1:L PR[91] R[100]mm/sec CNT100;
   1:  PR[91,1] = PR[90,1] + 1.228;
   1:L PR[91] R[100]mm/sec CNT100;
   1:  PR[91,1] = PR[90,1] + 2.241;
   1:  PR[91,2] = PR[90,2] + -13.861;
   1:L PR[91] R[100]mm/sec CNT100;
   1:  PR[91,1] = PR[90,1] + 2.519;
   1:  PR[91,2] = PR[90,2] + -14.188;
   1:L PR[91] R[100]mm/sec CNT100;
   1:  PR[91,1] = PR[90,1] + 4.490;
   1:  PR[91,2] = PR[90,2] + -15.923;
   1:L PR[91] R[100]mm/sec CNT100;
   1:  PR[91,1] = PR[90,1] + 6.006;
   1:  PR[91,2] = PR[90,2] + -16.894;
   1:L PR[91] R[100]mm/sec CNT100;
   1:  PR[91,1] = PR[90,1] + 6.840;
   1:  PR[91,2] = PR[90,2] + -17.469;
   1:L PR[91] R[100]mm/sec CNT100;
   1:  PR[91,1] = PR[90,1] + 10.686;
   1:  PR[91,2] = PR[90,2] + -19.130;
   1:L PR[91] R[100]mm/sec CNT100;
   1:  PR[91,1] = PR[90,1] + 13.082;
   1:  PR[91,2] = PR[90,2] + -19.752;
   1:L PR[91] R[100]mm/sec CNT100;
   1:  PR[91,1] = PR[90,1] + 15.994;
   1:  PR[91,2] = PR[90,2] + -20.057;
   1:L PR[91] R[100]mm/sec CNT100;
   1:  PR[91,1] = PR[90,1] + 17.091;
   1:  PR[91,2] = PR[90,2] + -20.209;
   1:L PR[91] R[100]mm/sec CNT100;
   1:  PR[91,1] = PR[90,1] + 20.020;
   1:  PR[91,2] = PR[90,2] + -20.057;
   1:L PR[91] R[100]mm/sec CNT100;
   1:  PR[91,1] = PR[90,1] + 20.730;
   1:  PR[91,2] = PR[90,2] + -19.975;
   1:L PR[91] R[100]mm/sec CNT100;
   1:  PR[91,1] = PR[90,1] + 23.699;
   1:  PR[91,2] = PR[90,2] + -19.360;
   1:L PR[91] R[100]mm/sec CNT100;
   1:  PR[91,1] = PR[90,1] + 26.996;
   1:  PR[91,2] = PR[90,2] + -18.139;
   1:L PR[91] R[100]mm/sec CNT100;
   1:  PR[91,1] = PR[90,1] + 29.867;
   1:  PR[91,2] = PR[90,2] + -16.549;
   1:L PR[91] R[100]mm/sec CNT100;
   1:  PR[91,1] = PR[90,1] + 30.115;
   1:  PR[91,2] = PR[90,2] + -16.340;
   1:L PR[91] R[100]mm/sec CNT100;
   1:  PR[91,1] = PR[90,1] + 32.699;
   1:  PR[91,2] = PR[90,2] + -14.301;
   1:L PR[91] R[100]mm/sec CNT100;
   1:  PR[91,1] = PR[90,1] + 34.384;
   1:  PR[91,2] = PR[90,2] + -12.492;
   1:L PR[91] R[100]mm/sec CNT100;
   1:  PR[91,1] = PR[90,1] + 35.168;
   1:  PR[91,2] = PR[90,2] + -11.397;
   1:L PR[91] R[100]mm/sec CNT100;
   1:  PR[91,1] = PR[90,1] + 36.471;
   1:  PR[91,2] = PR[90,2] + -9.425;
   1:L PR[91] R[100]mm/sec CNT100;
   1:  PR[91,1] = PR[90,1] + 37.308;
   1:  PR[91,2] = PR[90,2] + -7.571;
   1:L PR[91] R[100]mm/sec CNT100;
   1:  PR[91,1] = PR[90,1] + 37.992;
   1:  PR[91,2] = PR[90,2] + -5.876;
   1:L PR[91] R[100]mm/sec CNT100;
   1:  PR[91,1] = PR[90,1] + 38.438;
   1:  PR[91,2] = PR[90,2] + -4.177;
   1:L PR[91] R[100]mm/sec CNT100;
   1:  PR[91,1] = PR[90,1] + 38.700;
   1:  PR[91,2] = PR[90,2] + -2.102;
   1:L PR[91] R[100]mm/sec CNT100;
   1:  PR[91,1] = PR[90,1] + 38.842;
   1:  PR[91,2] = PR[90,2] + -0.345;
   1:L PR[91] R[100]mm/sec CNT100;
   1:  PR[91,1] = PR[90,1] + 38.580;
   1:  PR[91,2] = PR[90,2] + 1.712;
   1:L PR[91] R[100]mm/sec CNT100;
   1:  PR[91,1] = PR[90,1] + 38.429;
   1:  PR[91,2] = PR[90,2] + 3.585;
   1:L PR[91] R[100]mm/sec CNT100;
   1:  PR[91,1] = PR[90,1] + 37.992;
   1:  PR[91,2] = PR[90,2] + 5.253;
   1:L PR[91] R[100]mm/sec CNT100;
   1:  PR[91,1] = PR[90,1] + 37.308;
   1:  PR[91,2] = PR[90,2] + 6.948;
   1:L PR[91] R[100]mm/sec CNT100;
   1:  PR[91,1] = PR[90,1] + 36.483;
   1:  PR[91,2] = PR[90,2] + 8.775;
   1:L PR[91] R[100]mm/sec CNT100;
   1:  PR[91,1] = PR[90,1] + 35.589;
   1:  PR[91,2] = PR[90,2] + 10.016;
   1:L PR[91] R[100]mm/sec CNT100;
   1:  PR[91,1] = PR[90,1] + 34.362;
   1:  PR[91,2] = PR[90,2] + 11.891;
   1:L PR[91] R[100]mm/sec CNT100;
   1:  PR[91,1] = PR[90,1] + 32.681;
   1:  PR[91,2] = PR[90,2] + 13.697;
   1:L PR[91] R[100]mm/sec CNT100;
   1:  PR[91,1] = PR[90,1] + 32.064;
   1:  PR[91,2] = PR[90,2] + 14.222;
   1:L PR[91] R[100]mm/sec CNT100;
   1:  PR[91,1] = PR[90,1] + 29.892;
   1:  PR[91,2] = PR[90,2] + 15.911;
   1:L PR[91] R[100]mm/sec CNT100;
   1:  PR[91,1] = PR[90,1] + 26.997;
   1:  PR[91,2] = PR[90,2] + 17.515;
   1:L PR[91] R[100]mm/sec CNT100;
   1:  PR[91,1] = PR[90,1] + 23.702;
   1:  PR[91,2] = PR[90,2] + 18.735;
   1:L PR[91] R[100]mm/sec CNT100;
   1:  PR[91,1] = PR[90,1] + 20.734;
   1:  PR[91,2] = PR[90,2] + 19.350;
   1:L PR[91] R[100]mm/sec CNT100;
   1:  PR[91,1] = PR[90,1] + 20.026;
   1:  PR[91,2] = PR[90,2] + 19.433;
   1:L PR[91] R[100]mm/sec CNT100;
   1:  PR[91,1] = PR[90,1] + 17.073;
   1:  PR[91,2] = PR[90,2] + 19.587;
   1:L PR[91] R[100]mm/sec CNT100;
   1:  PR[91,1] = PR[90,1] + 14.440;
   1:  PR[91,2] = PR[90,2] + 19.320;
   1:L PR[91] R[100]mm/sec CNT100;
   1:  PR[91,1] = PR[90,1] + 13.118;
   1:  PR[91,2] = PR[90,2] + 19.137;
   1:L PR[91] R[100]mm/sec CNT100;
   1:  PR[91,1] = PR[90,1] + 10.704;
   1:  PR[91,2] = PR[90,2] + 18.511;
   1:L PR[91] R[100]mm/sec CNT100;
   1:  PR[91,1] = PR[90,1] + 8.577;
   1:  PR[91,2] = PR[90,2] + 17.581;
   1:L PR[91] R[100]mm/sec CNT100;
   1:  PR[91,1] = PR[90,1] + 6.863;
   1:  PR[91,2] = PR[90,2] + 16.864;
   1:L PR[91] R[100]mm/sec CNT100;
   1:  PR[91,1] = PR[90,1] + 5.059;
   1:  PR[91,2] = PR[90,2] + 15.713;
   1:L PR[91] R[100]mm/sec CNT100;
   1:  PR[91,1] = PR[90,1] + 4.729;
   1:  PR[91,2] = PR[90,2] + 15.485;
   1:L PR[91] R[100]mm/sec CNT100;
   1:  PR[91,1] = PR[90,1] + 4.115;
   1:  PR[91,2] = PR[90,2] + 14.999;
   1:L PR[91] R[100]mm/sec CNT100;
   1:  PR[91,1] = PR[90,1] + 2.650;
   1:  PR[91,2] = PR[90,2] + 13.694;
   1:L PR[91] R[100]mm/sec CNT100;
   1:  PR[91,1] = PR[90,1] + 2.187;
   1:  PR[91,2] = PR[90,2] + 13.207;
   1:L PR[91] R[100]mm/sec CNT100;
   1:  PR[91,1] = PR[90,1] + 2.071;
   1:  PR[91,2] = PR[90,2] + 13.124;
   1:L PR[91] R[100]mm/sec CNT100;
   1:  PR[91,1] = PR[90,1] + 1.975;
   1:  PR[91,2] = PR[90,2] + 12.997;
   1:L PR[91] R[100]mm/sec CNT100;
   1:  PR[91,1] = PR[90,1] + 1.492;
   1:  PR[91,2] = PR[90,2] + 12.655;
   1:L PR[91] R[100]mm/sec CNT100;
   1:  PR[91,1] = PR[90,1] + 0.659;
   1:  PR[91,2] = PR[90,2] + 12.199;
   1:L PR[91] R[100]mm/sec CNT100;
   1:  PR[91,1] = PR[90,1] + -0.537;
   1:L PR[91] R[100]mm/sec CNT100;
   1:  PR[91] = PR[90];
   1:  PR[91,1] = PR[90,1] + -1.619;
   1:  PR[91,2] = PR[90,2] + 13.007;
   1:  PR[91,3] = PR[90,3] + 29.585;
   1:L PR[91] R[100]mm/sec CNT100;
   1:  PR[91,1] = PR[90,1] + -2.026;
   1:  PR[91,2] = PR[90,2] + 13.535;
   1:L PR[91] R[100]mm/sec CNT100;
   1:  PR[91,1] = PR[90,1] + -2.284;
   1:  PR[91,2] = PR[90,2] + 13.796;
   1:L PR[91] R[100]mm/sec CNT100;
   1:  PR[91,1] = PR[90,1] + -3.663;
   1:  PR[91,2] = PR[90,2] + 15.020;
   1:L PR[91] R[100]mm/sec CNT100;
   1:  PR[91,1] = PR[90,1] + -4.322;
   1:  PR[91,2] = PR[90,2] + 15.541;
   1:L PR[91] R[100]mm/sec CNT100;
   1:  PR[91,1] = PR[90,1] + -5.881;
   1:  PR[91,2] = PR[90,2] + 16.540;
   1:L PR[91] R[100]mm/sec CNT100;
   1:  PR[91,1] = PR[90,1] + -6.447;
   1:  PR[91,2] = PR[90,2] + 16.919;
   1:L PR[91] R[100]mm/sec CNT100;
   1:  PR[91,1] = PR[90,1] + -8.547;
   1:  PR[91,2] = PR[90,2] + 17.837;
   1:L PR[91] R[100]mm/sec CNT100;
   1:  PR[91,1] = PR[90,1] + -10.347;
   1:  PR[91,2] = PR[90,2] + 18.591;
   1:L PR[91] R[100]mm/sec CNT100;
   1:  PR[91,1] = PR[90,1] + -12.616;
   1:  PR[91,2] = PR[90,2] + 19.178;
   1:L PR[91] R[100]mm/sec CNT100;
   1:  PR[91,1] = PR[90,1] + -15.383;
   1:  PR[91,2] = PR[90,2] + 19.466;
   1:L PR[91] R[100]mm/sec CNT100;
   1:  PR[91,1] = PR[90,1] + -16.726;
   1:  PR[91,2] = PR[90,2] + 19.649;
   1:L PR[91] R[100]mm/sec CNT100;
   1:  PR[91,1] = PR[90,1] + -19.525;
   1:  PR[91,2] = PR[90,2] + 19.502;
   1:L PR[91] R[100]mm/sec CNT100;
   1:  PR[91,1] = PR[90,1] + -20.474;
   1:  PR[91,2] = PR[90,2] + 19.389;
   1:L PR[91] R[100]mm/sec CNT100;
   1:  PR[91,1] = PR[90,1] + -23.312;
   1:  PR[91,2] = PR[90,2] + 18.800;
   1:L PR[91] R[100]mm/sec CNT100;
   1:  PR[91,1] = PR[90,1] + -26.695;
   1:  PR[91,2] = PR[90,2] + 17.538;
   1:L PR[91] R[100]mm/sec CNT100;
   1:  PR[91,1] = PR[90,1] + -29.547;
   1:  PR[91,2] = PR[90,2] + 15.940;
   1:L PR[91] R[100]mm/sec CNT100;
   1:  PR[91,1] = PR[90,1] + -32.277;
   1:  PR[91,2] = PR[90,2] + 13.788;
   1:L PR[91] R[100]mm/sec CNT100;
   1:  PR[91,1] = PR[90,1] + -34.179;
   1:  PR[91,2] = PR[90,2] + 11.741;
   1:L PR[91] R[100]mm/sec CNT100;
   1:  PR[91,1] = PR[90,1] + -34.665;
   1:  PR[91,2] = PR[90,2] + 11.063;
   1:L PR[91] R[100]mm/sec CNT100;
   1:  PR[91,1] = PR[90,1] + -36.145;
   1:  PR[91,2] = PR[90,2] + 8.811;
   1:L PR[91] R[100]mm/sec CNT100;
   1:  PR[91,1] = PR[90,1] + -37.114;
   1:  PR[91,2] = PR[90,2] + 6.635;
   1:L PR[91] R[100]mm/sec CNT100;
   1:  PR[91,1] = PR[90,1] + -37.627;
   1:  PR[91,2] = PR[90,2] + 5.357;
   1:L PR[91] R[100]mm/sec CNT100;
   1:  PR[91,1] = PR[90,1] + -38.150;
   1:  PR[91,2] = PR[90,2] + 3.335;
   1:L PR[91] R[100]mm/sec CNT100;
   1:  PR[91,1] = PR[90,1] + -38.352;
   1:  PR[91,2] = PR[90,2] + 1.744;
   1:L PR[91] R[100]mm/sec CNT100;
   1:  PR[91,1] = PR[90,1] + -38.512;
   1:  PR[91,2] = PR[90,2] + -0.277;
   1:L PR[91] R[100]mm/sec CNT100;
   1:  PR[91,1] = PR[90,1] + -38.308;
   1:  PR[91,2] = PR[90,2] + -1.869;
   1:L PR[91] R[100]mm/sec CNT100;
   1:  PR[91,1] = PR[90,1] + -38.141;
   1:  PR[91,2] = PR[90,2] + -3.993;
   1:L PR[91] R[100]mm/sec CNT100;
   1:  PR[91,1] = PR[90,1] + -37.627;
   1:  PR[91,2] = PR[90,2] + -5.981;
   1:L PR[91] R[100]mm/sec CNT100;
   1:  PR[91,1] = PR[90,1] + -37.114;
   1:  PR[91,2] = PR[90,2] + -7.260;
   1:L PR[91] R[100]mm/sec CNT100;
   1:  PR[91,1] = PR[90,1] + -36.157;
   1:  PR[91,2] = PR[90,2] + -9.406;
   1:L PR[91] R[100]mm/sec CNT100;
   1:  PR[91,1] = PR[90,1] + -35.527;
   1:  PR[91,2] = PR[90,2] + -10.281;
   1:L PR[91] R[100]mm/sec CNT100;
   1:  PR[91,1] = PR[90,1] + -34.157;
   1:  PR[91,2] = PR[90,2] + -12.389;
   1:L PR[91] R[100]mm/sec CNT100;
   1:  PR[91,1] = PR[90,1] + -32.259;
   1:  PR[91,2] = PR[90,2] + -14.431;
   1:L PR[91] R[100]mm/sec CNT100;
   1:  PR[91,1] = PR[90,1] + -32.014;
   1:  PR[91,2] = PR[90,2] + -14.638;
   1:L PR[91] R[100]mm/sec CNT100;
   1:  PR[91,1] = PR[90,1] + -29.550;
   1:  PR[91,2] = PR[90,2] + -16.562;
   1:L PR[91] R[100]mm/sec CNT100;
   1:  PR[91,1] = PR[90,1] + -26.695;
   1:  PR[91,2] = PR[90,2] + -18.162;
   1:L PR[91] R[100]mm/sec CNT100;
   1:  PR[91,1] = PR[90,1] + -23.839;
   1:  PR[91,2] = PR[90,2] + -19.216;
   1:L PR[91] R[100]mm/sec CNT100;
   1:  PR[91,1] = PR[90,1] + -23.297;
   1:  PR[91,2] = PR[90,2] + -19.428;
   1:L PR[91] R[100]mm/sec CNT100;
   1:  PR[91,1] = PR[90,1] + -20.469;
   1:  PR[91,2] = PR[90,2] + -20.015;
   1:L PR[91] R[100]mm/sec CNT100;
   1:  PR[91,1] = PR[90,1] + -19.518;
   1:  PR[91,2] = PR[90,2] + -20.125;
   1:L PR[91] R[100]mm/sec CNT100;
   1:  PR[91,1] = PR[90,1] + -16.690;
   1:  PR[91,2] = PR[90,2] + -20.275;
   1:L PR[91] R[100]mm/sec CNT100;
   1:  PR[91,1] = PR[90,1] + -14.178;
   1:  PR[91,2] = PR[90,2] + -20.022;
   1:L PR[91] R[100]mm/sec CNT100;
   1:  PR[91,1] = PR[90,1] + -12.625;
   1:  PR[91,2] = PR[90,2] + -19.804;
   1:L PR[91] R[100]mm/sec CNT100;
   1:  PR[91,1] = PR[90,1] + -10.342;
   1:  PR[91,2] = PR[90,2] + -19.214;
   1:L PR[91] R[100]mm/sec CNT100;
   1:  PR[91,1] = PR[90,1] + -8.326;
   1:  PR[91,2] = PR[90,2] + -18.330;
   1:L PR[91] R[100]mm/sec CNT100;
   1:  PR[91,1] = PR[90,1] + -6.368;
   1:  PR[91,2] = PR[90,2] + -17.495;
   1:L PR[91] R[100]mm/sec CNT100;
   1:  PR[91,1] = PR[90,1] + -4.682;
   1:  PR[91,2] = PR[90,2] + -16.417;
   1:L PR[91] R[100]mm/sec CNT100;
   1:  PR[91,1] = PR[90,1] + -4.107;
   1:  PR[91,2] = PR[90,2] + -16.003;
   1:L PR[91] R[100]mm/sec CNT100;
   1:  PR[91,1] = PR[90,1] + -2.186;
   1:  PR[91,2] = PR[90,2] + -14.321;
   1:L PR[91] R[100]mm/sec CNT100;
   1:  PR[91,1] = PR[90,1] + -2.028;
   1:  PR[91,2] = PR[90,2] + -14.158;
   1:L PR[91] R[100]mm/sec CNT100;
   1:  PR[91,1] = PR[90,1] + -1.445;
   1:  PR[91,2] = PR[90,2] + -13.690;
   1:L PR[91] R[100]mm/sec CNT100;
   1:  PR[91,1] = PR[90,1] + -0.428;
   1:  PR[91,2] = PR[90,2] + -12.971;
   1:L PR[91] R[100]mm/sec CNT100;
   1:  PR[91,1] = PR[90,1] + 0.811;
   1:  PR[91,2] = PR[90,2] + -13.411;
   1:L PR[91] R[100]mm/sec CNT100;
   1:  PR[91,1] = PR[90,1] + 1.263;
   1:L PR[91] R[100]mm/sec CNT100;
   1:  PR[91,1] = PR[90,1] + 2.190;
   1:  PR[91,2] = PR[90,2] + -14.163;
   1:L PR[91] R[100]mm/sec CNT100;
   1:  PR[91,1] = PR[90,1] + 2.348;
   1:  PR[91,2] = PR[90,2] + -14.325;
   1:L PR[91] R[100]mm/sec CNT100;
   1:  PR[91,1] = PR[90,1] + 4.243;
   1:  PR[91,2] = PR[90,2] + -15.987;
   1:L PR[91] R[100]mm/sec CNT100;
   1:  PR[91,1] = PR[90,1] + 5.610;
   1:  PR[91,2] = PR[90,2] + -16.862;
   1:L PR[91] R[100]mm/sec CNT100;
   1:  PR[91,1] = PR[90,1] + 6.547;
   1:  PR[91,2] = PR[90,2] + -17.508;
   1:L PR[91] R[100]mm/sec CNT100;
   1:  PR[91,1] = PR[90,1] + 10.488;
   1:  PR[91,2] = PR[90,2] + -19.209;
   1:L PR[91] R[100]mm/sec CNT100;
   1:  PR[91,1] = PR[90,1] + 12.755;
   1:  PR[91,2] = PR[90,2] + -19.796;
   1:L PR[91] R[100]mm/sec CNT100;
   1:  PR[91,1] = PR[90,1] + 15.518;
   1:  PR[91,2] = PR[90,2] + -20.086;
   1:L PR[91] R[100]mm/sec CNT100;
   1:  PR[91,1] = PR[90,1] + 16.865;
   1:  PR[91,2] = PR[90,2] + -20.273;
   1:L PR[91] R[100]mm/sec CNT100;
   1:  PR[91,1] = PR[90,1] + 19.652;
   1:  PR[91,2] = PR[90,2] + -20.129;
   1:L PR[91] R[100]mm/sec CNT100;
   1:  PR[91,1] = PR[90,1] + 20.605;
   1:  PR[91,2] = PR[90,2] + -20.018;
   1:L PR[91] R[100]mm/sec CNT100;
   1:  PR[91,1] = PR[90,1] + 23.441;
   1:  PR[91,2] = PR[90,2] + -19.431;
   1:L PR[91] R[100]mm/sec CNT100;
   1:  PR[91,1] = PR[90,1] + 26.553;
   1:  PR[91,2] = PR[90,2] + -18.281;
   1:L PR[91] R[100]mm/sec CNT100;
   1:  PR[91,1] = PR[90,1] + 26.823;
   1:  PR[91,2] = PR[90,2] + -18.176;
   1:L PR[91] R[100]mm/sec CNT100;
   1:  PR[91,1] = PR[90,1] + 29.673;
   1:  PR[91,2] = PR[90,2] + -16.588;
   1:L PR[91] R[100]mm/sec CNT100;
   1:  PR[91,1] = PR[90,1] + 32.387;
   1:  PR[91,2] = PR[90,2] + -14.456;
   1:L PR[91] R[100]mm/sec CNT100;
   1:  PR[91,1] = PR[90,1] + 34.304;
   1:  PR[91,2] = PR[90,2] + -12.397;
   1:L PR[91] R[100]mm/sec CNT100;
   1:  PR[91,1] = PR[90,1] + 34.787;
   1:  PR[91,2] = PR[90,2] + -11.722;
   1:L PR[91] R[100]mm/sec CNT100;
   1:  PR[91,1] = PR[90,1] + 36.293;
   1:  PR[91,2] = PR[90,2] + -9.444;
   1:L PR[91] R[100]mm/sec CNT100;
   1:  PR[91,1] = PR[90,1] + 37.261;
   1:  PR[91,2] = PR[90,2] + -7.300;
   1:L PR[91] R[100]mm/sec CNT100;
   1:  PR[91,1] = PR[90,1] + 37.773;
   1:  PR[91,2] = PR[90,2] + -6.031;
   1:L PR[91] R[100]mm/sec CNT100;
   1:  PR[91,1] = PR[90,1] + 38.297;
   1:  PR[91,2] = PR[90,2] + -4.030;
   1:L PR[91] R[100]mm/sec CNT100;
   1:  PR[91,1] = PR[90,1] + 38.499;
   1:  PR[91,2] = PR[90,2] + -2.435;
   1:L PR[91] R[100]mm/sec CNT100;
   1:  PR[91,1] = PR[90,1] + 38.668;
   1:  PR[91,2] = PR[90,2] + -0.345;
   1:L PR[91] R[100]mm/sec CNT100;
   1:  PR[91,1] = PR[90,1] + 38.465;
   1:  PR[91,2] = PR[90,2] + 1.250;
   1:L PR[91] R[100]mm/sec CNT100;
   1:  PR[91,1] = PR[90,1] + 38.289;
   1:  PR[91,2] = PR[90,2] + 3.439;
   1:L PR[91] R[100]mm/sec CNT100;
   1:  PR[91,1] = PR[90,1] + 37.773;
   1:  PR[91,2] = PR[90,2] + 5.408;
   1:L PR[91] R[100]mm/sec CNT100;
   1:  PR[91,1] = PR[90,1] + 37.260;
   1:  PR[91,2] = PR[90,2] + 6.676;
   1:L PR[91] R[100]mm/sec CNT100;
   1:  PR[91,1] = PR[90,1] + 36.304;
   1:  PR[91,2] = PR[90,2] + 8.794;
   1:L PR[91] R[100]mm/sec CNT100;
   1:  PR[91,1] = PR[90,1] + 35.674;
   1:  PR[91,2] = PR[90,2] + 9.669;
   1:L PR[91] R[100]mm/sec CNT100;
   1:  PR[91,1] = PR[90,1] + 34.283;
   1:  PR[91,2] = PR[90,2] + 11.796;
   1:L PR[91] R[100]mm/sec CNT100;
   1:  PR[91,1] = PR[90,1] + 32.368;
   1:  PR[91,2] = PR[90,2] + 13.853;
   1:L PR[91] R[100]mm/sec CNT100;
   1:  PR[91,1] = PR[90,1] + 32.130;
   1:  PR[91,2] = PR[90,2] + 14.055;
   1:L PR[91] R[100]mm/sec CNT100;
   1:  PR[91,1] = PR[90,1] + 29.677;
   1:  PR[91,2] = PR[90,2] + 15.962;
   1:L PR[91] R[100]mm/sec CNT100;
   1:  PR[91,1] = PR[90,1] + 26.836;
   1:  PR[91,2] = PR[90,2] + 17.544;
   1:L PR[91] R[100]mm/sec CNT100;
   1:  PR[91,1] = PR[90,1] + 23.975;
   1:  PR[91,2] = PR[90,2] + 18.596;
   1:L PR[91] R[100]mm/sec CNT100;
   1:  PR[91,1] = PR[90,1] + 23.432;
   1:  PR[91,2] = PR[90,2] + 18.808;
   1:L PR[91] R[100]mm/sec CNT100;
   1:  PR[91,1] = PR[90,1] + 20.609;
   1:  PR[91,2] = PR[90,2] + 19.392;
   1:L PR[91] R[100]mm/sec CNT100;
   1:  PR[91,1] = PR[90,1] + 19.659;
   1:  PR[91,2] = PR[90,2] + 19.505;
   1:L PR[91] R[100]mm/sec CNT100;
   1:  PR[91,1] = PR[90,1] + 16.849;
   1:  PR[91,2] = PR[90,2] + 19.651;
   1:L PR[91] R[100]mm/sec CNT100;
   1:  PR[91,1] = PR[90,1] + 14.343;
   1:  PR[91,2] = PR[90,2] + 19.397;
   1:L PR[91] R[100]mm/sec CNT100;
   1:  PR[91,1] = PR[90,1] + 12.793;
   1:  PR[91,2] = PR[90,2] + 19.182;
   1:L PR[91] R[100]mm/sec CNT100;
   1:  PR[91,1] = PR[90,1] + 10.508;
   1:  PR[91,2] = PR[90,2] + 18.590;
   1:L PR[91] R[100]mm/sec CNT100;
   1:  PR[91,1] = PR[90,1] + 8.492;
   1:  PR[91,2] = PR[90,2] + 17.708;
   1:L PR[91] R[100]mm/sec CNT100;
   1:  PR[91,1] = PR[90,1] + 6.576;
   1:  PR[91,2] = PR[90,2] + 16.907;
   1:L PR[91] R[100]mm/sec CNT100;
   1:  PR[91,1] = PR[90,1] + 4.877;
   1:  PR[91,2] = PR[90,2] + 15.823;
   1:L PR[91] R[100]mm/sec CNT100;
   1:  PR[91,1] = PR[90,1] + 4.508;
   1:  PR[91,2] = PR[90,2] + 15.568;
   1:L PR[91] R[100]mm/sec CNT100;
   1:  PR[91,1] = PR[90,1] + 3.827;
   1:  PR[91,2] = PR[90,2] + 15.029;
   1:L PR[91] R[100]mm/sec CNT100;
   1:  PR[91,1] = PR[90,1] + 2.455;
   1:  PR[91,2] = PR[90,2] + 13.810;
   1:L PR[91] R[100]mm/sec CNT100;
   1:  PR[91,1] = PR[90,1] + 2.167;
   1:  PR[91,2] = PR[90,2] + 13.507;
   1:L PR[91] R[100]mm/sec CNT100;
   1:  PR[91,1] = PR[90,1] + 1.982;
   1:  PR[91,2] = PR[90,2] + 13.374;
   1:L PR[91] R[100]mm/sec CNT100;
   1:  PR[91,1] = PR[90,1] + 1.918;
   1:  PR[91,2] = PR[90,2] + 13.290;
   1:L PR[91] R[100]mm/sec CNT100;
   1:  PR[91,1] = PR[90,1] + 1.516;
   1:  PR[91,2] = PR[90,2] + 13.005;
   1:L PR[91] R[100]mm/sec CNT100;
   1:  PR[91,1] = PR[90,1] + 0.619;
   1:  PR[91,2] = PR[90,2] + 12.514;
   1:L PR[91] R[100]mm/sec CNT100;
   1:  PR[91,1] = PR[90,1] + -0.513;
   1:L PR[91] R[100]mm/sec CNT100;
   1:  PR[91] = PR[90];
   1:  PR[91,1] = PR[90,1] + -1.659;
   1:  PR[91,2] = PR[90,2] + 13.350;
   1:  PR[91,3] = PR[90,3] + 30.195;
   1:L PR[91] R[100]mm/sec CNT100;
   1:  PR[91,1] = PR[90,1] + -2.094;
   1:  PR[91,2] = PR[90,2] + 13.916;
   1:L PR[91] R[100]mm/sec CNT100;
   1:  PR[91,1] = PR[90,1] + -3.375;
   1:  PR[91,2] = PR[90,2] + 15.051;
   1:L PR[91] R[100]mm/sec CNT100;
   1:  PR[91,1] = PR[90,1] + -4.102;
   1:  PR[91,2] = PR[90,2] + 15.625;
   1:L PR[91] R[100]mm/sec CNT100;
   1:  PR[91,1] = PR[90,1] + -5.528;
   1:  PR[91,2] = PR[90,2] + 16.538;
   1:L PR[91] R[100]mm/sec CNT100;
   1:  PR[91,1] = PR[90,1] + -6.160;
   1:  PR[91,2] = PR[90,2] + 16.962;
   1:L PR[91] R[100]mm/sec CNT100;
   1:  PR[91,1] = PR[90,1] + -8.132;
   1:  PR[91,2] = PR[90,2] + 17.824;
   1:L PR[91] R[100]mm/sec CNT100;
   1:  PR[91,1] = PR[90,1] + -10.152;
   1:  PR[91,2] = PR[90,2] + 18.670;
   1:L PR[91] R[100]mm/sec CNT100;
   1:  PR[91,1] = PR[90,1] + -12.291;
   1:  PR[91,2] = PR[90,2] + 19.223;
   1:L PR[91] R[100]mm/sec CNT100;
   1:  PR[91,1] = PR[90,1] + -14.909;
   1:  PR[91,2] = PR[90,2] + 19.496;
   1:L PR[91] R[100]mm/sec CNT100;
   1:  PR[91,1] = PR[90,1] + -16.502;
   1:  PR[91,2] = PR[90,2] + 19.713;
   1:L PR[91] R[100]mm/sec CNT100;
   1:  PR[91,1] = PR[90,1] + -19.158;
   1:  PR[91,2] = PR[90,2] + 19.573;
   1:L PR[91] R[100]mm/sec CNT100;
   1:  PR[91,1] = PR[90,1] + -20.349;
   1:  PR[91,2] = PR[90,2] + 19.432;
   1:L PR[91] R[100]mm/sec CNT100;
   1:  PR[91,1] = PR[90,1] + -23.053;
   1:  PR[91,2] = PR[90,2] + 18.871;
   1:L PR[91] R[100]mm/sec CNT100;
   1:  PR[91,1] = PR[90,1] + -26.533;
   1:  PR[91,2] = PR[90,2] + 17.568;
   1:L PR[91] R[100]mm/sec CNT100;
   1:  PR[91,1] = PR[90,1] + -29.264;
   1:  PR[91,2] = PR[90,2] + 16.038;
   1:L PR[91] R[100]mm/sec CNT100;
   1:  PR[91,1] = PR[90,1] + -31.985;
   1:  PR[91,2] = PR[90,2] + 13.921;
   1:L PR[91] R[100]mm/sec CNT100;
   1:  PR[91,1] = PR[90,1] + -34.103;
   1:  PR[91,2] = PR[90,2] + 11.641;
   1:L PR[91] R[100]mm/sec CNT100;
   1:  PR[91,1] = PR[90,1] + -34.288;
   1:  PR[91,2] = PR[90,2] + 11.383;
   1:L PR[91] R[100]mm/sec CNT100;
   1:  PR[91,1] = PR[90,1] + -35.967;
   1:  PR[91,2] = PR[90,2] + 8.828;
   1:L PR[91] R[100]mm/sec CNT100;
   1:  PR[91,1] = PR[90,1] + -37.068;
   1:  PR[91,2] = PR[90,2] + 6.358;
   1:L PR[91] R[100]mm/sec CNT100;
   1:  PR[91,1] = PR[90,1] + -37.409;
   1:  PR[91,2] = PR[90,2] + 5.507;
   1:L PR[91] R[100]mm/sec CNT100;
   1:  PR[91,1] = PR[90,1] + -38.011;
   1:  PR[91,2] = PR[90,2] + 3.181;
   1:L PR[91] R[100]mm/sec CNT100;
   1:  PR[91,1] = PR[90,1] + -38.152;
   1:  PR[91,2] = PR[90,2] + 2.067;
   1:L PR[91] R[100]mm/sec CNT100;
   1:  PR[91,1] = PR[90,1] + -38.338;
   1:  PR[91,2] = PR[90,2] + -0.277;
   1:L PR[91] R[100]mm/sec CNT100;
   1:  PR[91,1] = PR[90,1] + -38.193;
   1:  PR[91,2] = PR[90,2] + -1.409;
   1:L PR[91] R[100]mm/sec CNT100;
   1:  PR[91,1] = PR[90,1] + -38.002;
   1:  PR[91,2] = PR[90,2] + -3.839;
   1:L PR[91] R[100]mm/sec CNT100;
   1:  PR[91,1] = PR[90,1] + -37.409;
   1:  PR[91,2] = PR[90,2] + -6.131;
   1:L PR[91] R[100]mm/sec CNT100;
   1:  PR[91,1] = PR[90,1] + -37.068;
   1:  PR[91,2] = PR[90,2] + -6.982;
   1:L PR[91] R[100]mm/sec CNT100;
   1:  PR[91,1] = PR[90,1] + -35.980;
   1:  PR[91,2] = PR[90,2] + -9.423;
   1:L PR[91] R[100]mm/sec CNT100;
   1:  PR[91,1] = PR[90,1] + -35.613;
   1:  PR[91,2] = PR[90,2] + -9.933;
   1:L PR[91] R[100]mm/sec CNT100;
   1:  PR[91,1] = PR[90,1] + -34.081;
   1:  PR[91,2] = PR[90,2] + -12.289;
   1:L PR[91] R[100]mm/sec CNT100;
   1:  PR[91,1] = PR[90,1] + -31.984;
   1:  PR[91,2] = PR[90,2] + -14.547;
   1:L PR[91] R[100]mm/sec CNT100;
   1:  PR[91,1] = PR[90,1] + -29.447;
   1:  PR[91,2] = PR[90,2] + -16.533;
   1:L PR[91] R[100]mm/sec CNT100;
   1:  PR[91,1] = PR[90,1] + -29.283;
   1:  PR[91,2] = PR[90,2] + -16.651;
   1:L PR[91] R[100]mm/sec CNT100;
   1:  PR[91,1] = PR[90,1] + -26.533;
   1:  PR[91,2] = PR[90,2] + -18.192;
   1:L PR[91] R[100]mm/sec CNT100;
   1:  PR[91,1] = PR[90,1] + -23.799;
   1:  PR[91,2] = PR[90,2] + -19.202;
   1:L PR[91] R[100]mm/sec CNT100;
   1:  PR[91,1] = PR[90,1] + -23.037;
   1:  PR[91,2] = PR[90,2] + -19.499;
   1:L PR[91] R[100]mm/sec CNT100;
   1:  PR[91,1] = PR[90,1] + -20.342;
   1:  PR[91,2] = PR[90,2] + -20.058;
   1:L PR[91] R[100]mm/sec CNT100;
   1:  PR[91,1] = PR[90,1] + -19.149;
   1:  PR[91,2] = PR[90,2] + -20.197;
   1:L PR[91] R[100]mm/sec CNT100;
   1:  PR[91,1] = PR[90,1] + -16.464;
   1:  PR[91,2] = PR[90,2] + -20.339;
   1:L PR[91] R[100]mm/sec CNT100;
   1:  PR[91,1] = PR[90,1] + -14.079;
   1:  PR[91,2] = PR[90,2] + -20.098;
   1:L PR[91] R[100]mm/sec CNT100;
   1:  PR[91,1] = PR[90,1] + -12.298;
   1:  PR[91,2] = PR[90,2] + -19.849;
   1:L PR[91] R[100]mm/sec CNT100;
   1:  PR[91,1] = PR[90,1] + -10.145;
   1:  PR[91,2] = PR[90,2] + -19.292;
   1:L PR[91] R[100]mm/sec CNT100;
   1:  PR[91,1] = PR[90,1] + -8.239;
   1:  PR[91,2] = PR[90,2] + -18.456;
   1:L PR[91] R[100]mm/sec CNT100;
   1:  PR[91,1] = PR[90,1] + -6.075;
   1:  PR[91,2] = PR[90,2] + -17.534;
   1:L PR[91] R[100]mm/sec CNT100;
   1:  PR[91,1] = PR[90,1] + -4.497;
   1:  PR[91,2] = PR[90,2] + -16.525;
   1:L PR[91] R[100]mm/sec CNT100;
   1:  PR[91,1] = PR[90,1] + -3.863;
   1:  PR[91,2] = PR[90,2] + -16.068;
   1:L PR[91] R[100]mm/sec CNT100;
   1:  PR[91,1] = PR[90,1] + -1.774;
   1:  PR[91,2] = PR[90,2] + -14.239;
   1:L PR[91] R[100]mm/sec CNT100;
   1:  PR[91,1] = PR[90,1] + -1.656;
   1:  PR[91,2] = PR[90,2] + -14.199;
   1:L PR[91] R[100]mm/sec CNT100;
   1:  PR[91,1] = PR[90,1] + -1.368;
   1:  PR[91,2] = PR[90,2] + -13.968;
   1:L PR[91] R[100]mm/sec CNT100;
   1:  PR[91,1] = PR[90,1] + -0.403;
   1:  PR[91,2] = PR[90,2] + -13.286;
   1:L PR[91] R[100]mm/sec CNT100;
   1:  PR[91,1] = PR[90,1] + 0.934;
   1:  PR[91,2] = PR[90,2] + -13.761;
   1:L PR[91] R[100]mm/sec CNT100;
   1:  PR[91,1] = PR[90,1] + 1.291;
   1:L PR[91] R[100]mm/sec CNT100;
   1:  PR[91,1] = PR[90,1] + 1.872;
   1:  PR[91,2] = PR[90,2] + -14.236;
   1:L PR[91] R[100]mm/sec CNT100;
   1:  PR[91,1] = PR[90,1] + 2.053;
   1:  PR[91,2] = PR[90,2] + -14.346;
   1:L PR[91] R[100]mm/sec CNT100;
   1:  PR[91,1] = PR[90,1] + 3.998;
   1:  PR[91,2] = PR[90,2] + -16.051;
   1:L PR[91] R[100]mm/sec CNT100;
   1:  PR[91,1] = PR[90,1] + 5.213;
   1:  PR[91,2] = PR[90,2] + -16.830;
   1:L PR[91] R[100]mm/sec CNT100;
   1:  PR[91,1] = PR[90,1] + 6.256;
   1:  PR[91,2] = PR[90,2] + -17.548;
   1:L PR[91] R[100]mm/sec CNT100;
   1:  PR[91,1] = PR[90,1] + 8.196;
   1:  PR[91,2] = PR[90,2] + -18.395;
   1:L PR[91] R[100]mm/sec CNT100;
   1:  PR[91,1] = PR[90,1] + 10.288;
   1:  PR[91,2] = PR[90,2] + -19.286;
   1:L PR[91] R[100]mm/sec CNT100;
   1:  PR[91,1] = PR[90,1] + 12.428;
   1:  PR[91,2] = PR[90,2] + -19.841;
   1:L PR[91] R[100]mm/sec CNT100;
   1:  PR[91,1] = PR[90,1] + 15.043;
   1:  PR[91,2] = PR[90,2] + -20.115;
   1:L PR[91] R[100]mm/sec CNT100;
   1:  PR[91,1] = PR[90,1] + 16.640;
   1:  PR[91,2] = PR[90,2] + -20.337;
   1:L PR[91] R[100]mm/sec CNT100;
   1:  PR[91,1] = PR[90,1] + 19.284;
   1:  PR[91,2] = PR[90,2] + -20.200;
   1:L PR[91] R[100]mm/sec CNT100;
   1:  PR[91,1] = PR[90,1] + 20.479;
   1:  PR[91,2] = PR[90,2] + -20.061;
   1:L PR[91] R[100]mm/sec CNT100;
   1:  PR[91,1] = PR[90,1] + 23.182;
   1:  PR[91,2] = PR[90,2] + -19.501;
   1:L PR[91] R[100]mm/sec CNT100;
   1:  PR[91,1] = PR[90,1] + 26.151;
   1:  PR[91,2] = PR[90,2] + -18.405;
   1:L PR[91] R[100]mm/sec CNT100;
   1:  PR[91,1] = PR[90,1] + 26.661;
   1:  PR[91,2] = PR[90,2] + -18.206;
   1:L PR[91] R[100]mm/sec CNT100;
   1:  PR[91,1] = PR[90,1] + 29.390;
   1:  PR[91,2] = PR[90,2] + -16.686;
   1:L PR[91] R[100]mm/sec CNT100;
   1:  PR[91,1] = PR[90,1] + 32.093;
   1:  PR[91,2] = PR[90,2] + -14.592;
   1:L PR[91] R[100]mm/sec CNT100;
   1:  PR[91,1] = PR[90,1] + 34.224;
   1:  PR[91,2] = PR[90,2] + -12.301;
   1:L PR[91] R[100]mm/sec CNT100;
   1:  PR[91,1] = PR[90,1] + 34.406;
   1:  PR[91,2] = PR[90,2] + -12.048;
   1:L PR[91] R[100]mm/sec CNT100;
   1:  PR[91,1] = PR[90,1] + 36.114;
   1:  PR[91,2] = PR[90,2] + -9.464;
   1:L PR[91] R[100]mm/sec CNT100;
   1:  PR[91,1] = PR[90,1] + 37.213;
   1:  PR[91,2] = PR[90,2] + -7.029;
   1:L PR[91] R[100]mm/sec CNT100;
   1:  PR[91,1] = PR[90,1] + 37.553;
   1:  PR[91,2] = PR[90,2] + -6.186;
   1:L PR[91] R[100]mm/sec CNT100;
   1:  PR[91,1] = PR[90,1] + 38.157;
   1:  PR[91,2] = PR[90,2] + -3.884;
   1:L PR[91] R[100]mm/sec CNT100;
   1:  PR[91,1] = PR[90,1] + 38.298;
   1:  PR[91,2] = PR[90,2] + -2.768;
   1:L PR[91] R[100]mm/sec CNT100;
   1:  PR[91,1] = PR[90,1] + 38.494;
   1:  PR[91,2] = PR[90,2] + -0.345;
   1:L PR[91] R[100]mm/sec CNT100;
   1:  PR[91,1] = PR[90,1] + 38.350;
   1:  PR[91,2] = PR[90,2] + 0.789;
   1:L PR[91] R[100]mm/sec CNT100;
   1:  PR[91,1] = PR[90,1] + 38.148;
   1:  PR[91,2] = PR[90,2] + 3.292;
   1:L PR[91] R[100]mm/sec CNT100;
   1:  PR[91,1] = PR[90,1] + 37.553;
   1:  PR[91,2] = PR[90,2] + 5.562;
   1:L PR[91] R[100]mm/sec CNT100;
   1:  PR[91,1] = PR[90,1] + 37.213;
   1:  PR[91,2] = PR[90,2] + 6.405;
   1:L PR[91] R[100]mm/sec CNT100;
   1:  PR[91,1] = PR[90,1] + 36.126;
   1:  PR[91,2] = PR[90,2] + 8.814;
   1:L PR[91] R[100]mm/sec CNT100;
   1:  PR[91,1] = PR[90,1] + 35.759;
   1:  PR[91,2] = PR[90,2] + 9.323;
   1:L PR[91] R[100]mm/sec CNT100;
   1:  PR[91,1] = PR[90,1] + 34.203;
   1:  PR[91,2] = PR[90,2] + 11.700;
   1:L PR[91] R[100]mm/sec CNT100;
   1:  PR[91,1] = PR[90,1] + 32.093;
   1:  PR[91,2] = PR[90,2] + 13.968;
   1:L PR[91] R[100]mm/sec CNT100;
   1:  PR[91,1] = PR[90,1] + 29.391;
   1:  PR[91,2] = PR[90,2] + 16.061;
   1:L PR[91] R[100]mm/sec CNT100;
   1:  PR[91,1] = PR[90,1] + 26.675;
   1:  PR[91,2] = PR[90,2] + 17.574;
   1:L PR[91] R[100]mm/sec CNT100;
   1:  PR[91,1] = PR[90,1] + 23.937;
   1:  PR[91,2] = PR[90,2] + 18.580;
   1:L PR[91] R[100]mm/sec CNT100;
   1:  PR[91,1] = PR[90,1] + 23.175;
   1:  PR[91,2] = PR[90,2] + 18.879;
   1:L PR[91] R[100]mm/sec CNT100;
   1:  PR[91,1] = PR[90,1] + 20.485;
   1:  PR[91,2] = PR[90,2] + 19.435;
   1:L PR[91] R[100]mm/sec CNT100;
   1:  PR[91,1] = PR[90,1] + 19.293;
   1:  PR[91,2] = PR[90,2] + 19.576;
   1:L PR[91] R[100]mm/sec CNT100;
   1:  PR[91,1] = PR[90,1] + 16.625;
   1:  PR[91,2] = PR[90,2] + 19.715;
   1:L PR[91] R[100]mm/sec CNT100;
   1:  PR[91,1] = PR[90,1] + 14.246;
   1:  PR[91,2] = PR[90,2] + 19.474;
   1:L PR[91] R[100]mm/sec CNT100;
   1:  PR[91,1] = PR[90,1] + 12.468;
   1:  PR[91,2] = PR[90,2] + 19.228;
   1:L PR[91] R[100]mm/sec CNT100;
   1:  PR[91,1] = PR[90,1] + 10.313;
   1:  PR[91,2] = PR[90,2] + 18.669;
   1:L PR[91] R[100]mm/sec CNT100;
   1:  PR[91,1] = PR[90,1] + 8.406;
   1:  PR[91,2] = PR[90,2] + 17.835;
   1:L PR[91] R[100]mm/sec CNT100;
   1:  PR[91,1] = PR[90,1] + 6.288;
   1:  PR[91,2] = PR[90,2] + 16.950;
   1:L PR[91] R[100]mm/sec CNT100;
   1:  PR[91,1] = PR[90,1] + 4.694;
   1:  PR[91,2] = PR[90,2] + 15.932;
   1:L PR[91] R[100]mm/sec CNT100;
   1:  PR[91,1] = PR[90,1] + 4.288;
   1:  PR[91,2] = PR[90,2] + 15.651;
   1:L PR[91] R[100]mm/sec CNT100;
   1:  PR[91,1] = PR[90,1] + 3.541;
   1:  PR[91,2] = PR[90,2] + 15.060;
   1:L PR[91] R[100]mm/sec CNT100;
   1:  PR[91,1] = PR[90,1] + 2.114;
   1:  PR[91,2] = PR[90,2] + 13.785;
   1:L PR[91] R[100]mm/sec CNT100;
   1:  PR[91,1] = PR[90,1] + 1.561;
   1:  PR[91,2] = PR[90,2] + 13.366;
   1:L PR[91] R[100]mm/sec CNT100;
   1:  PR[91,1] = PR[90,1] + 0.579;
   1:  PR[91,2] = PR[90,2] + 12.829;
   1:L PR[91] R[100]mm/sec CNT100;
   1:  PR[91,1] = PR[90,1] + -0.489;
   1:L PR[91] R[100]mm/sec CNT100;
   1:  PR[91] = PR[90];
   1:  PR[91,1] = PR[90,1] + -1.698;
   1:  PR[91,2] = PR[90,2] + 13.693;
   1:  PR[91,3] = PR[90,3] + 30.805;
   1:L PR[91] R[100]mm/sec CNT100;
   1:  PR[91,1] = PR[90,1] + -2.079;
   1:  PR[91,2] = PR[90,2] + 14.189;
   1:L PR[91] R[100]mm/sec CNT100;
   1:  PR[91,1] = PR[90,1] + -3.089;
   1:  PR[91,2] = PR[90,2] + 15.082;
   1:L PR[91] R[100]mm/sec CNT100;
   1:  PR[91,1] = PR[90,1] + -3.882;
   1:  PR[91,2] = PR[90,2] + 15.709;
   1:L PR[91] R[100]mm/sec CNT100;
   1:  PR[91,1] = PR[90,1] + -5.175;
   1:  PR[91,2] = PR[90,2] + 16.537;
   1:L PR[91] R[100]mm/sec CNT100;
   1:  PR[91,1] = PR[90,1] + -5.873;
   1:  PR[91,2] = PR[90,2] + 17.005;
   1:L PR[91] R[100]mm/sec CNT100;
   1:  PR[91,1] = PR[90,1] + -7.717;
   1:  PR[91,2] = PR[90,2] + 17.811;
   1:L PR[91] R[100]mm/sec CNT100;
   1:  PR[91,1] = PR[90,1] + -9.956;
   1:  PR[91,2] = PR[90,2] + 18.749;
   1:L PR[91] R[100]mm/sec CNT100;
   1:  PR[91,1] = PR[90,1] + -11.966;
   1:  PR[91,2] = PR[90,2] + 19.269;
   1:L PR[91] R[100]mm/sec CNT100;
   1:  PR[91,1] = PR[90,1] + -14.435;
   1:  PR[91,2] = PR[90,2] + 19.526;
   1:L PR[91] R[100]mm/sec CNT100;
   1:  PR[91,1] = PR[90,1] + -16.278;
   1:  PR[91,2] = PR[90,2] + 19.777;
   1:L PR[91] R[100]mm/sec CNT100;
   1:  PR[91,1] = PR[90,1] + -18.791;
   1:  PR[91,2] = PR[90,2] + 19.645;
   1:L PR[91] R[100]mm/sec CNT100;
   1:  PR[91,1] = PR[90,1] + -20.224;
   1:  PR[91,2] = PR[90,2] + 19.475;
   1:L PR[91] R[100]mm/sec CNT100;
   1:  PR[91,1] = PR[90,1] + -22.797;
   1:  PR[91,2] = PR[90,2] + 18.941;
   1:L PR[91] R[100]mm/sec CNT100;
   1:  PR[91,1] = PR[90,1] + -25.617;
   1:  PR[91,2] = PR[90,2] + 17.895;
   1:L PR[91] R[100]mm/sec CNT100;
   1:  PR[91,1] = PR[90,1] + -26.362;
   1:  PR[91,2] = PR[90,2] + 17.603;
   1:L PR[91] R[100]mm/sec CNT100;
   1:  PR[91,1] = PR[90,1] + -28.977;
   1:  PR[91,2] = PR[90,2] + 16.138;
   1:L PR[91] R[100]mm/sec CNT100;
   1:  PR[91,1] = PR[90,1] + -31.789;
   1:  PR[91,2] = PR[90,2] + 13.961;
   1:L PR[91] R[100]mm/sec CNT100;
   1:  PR[91,1] = PR[90,1] + -33.974;
   1:  PR[91,2] = PR[90,2] + 11.601;
   1:L PR[91] R[100]mm/sec CNT100;
   1:  PR[91,1] = PR[90,1] + -35.790;
   1:  PR[91,2] = PR[90,2] + 8.844;
   1:L PR[91] R[100]mm/sec CNT100;
   1:  PR[91,1] = PR[90,1] + -37.022;
   1:  PR[91,2] = PR[90,2] + 6.081;
   1:L PR[91] R[100]mm/sec CNT100;
   1:  PR[91,1] = PR[90,1] + -37.192;
   1:  PR[91,2] = PR[90,2] + 5.657;
   1:L PR[91] R[100]mm/sec CNT100;
   1:  PR[91,1] = PR[90,1] + -37.872;
   1:  PR[91,2] = PR[90,2] + 3.028;
   1:L PR[91] R[100]mm/sec CNT100;
   1:  PR[91,1] = PR[90,1] + -37.953;
   1:  PR[91,2] = PR[90,2] + 2.390;
   1:L PR[91] R[100]mm/sec CNT100;
   1:  PR[91,1] = PR[90,1] + -38.164;
   1:  PR[91,2] = PR[90,2] + -0.277;
   1:L PR[91] R[100]mm/sec CNT100;
   1:  PR[91,1] = PR[90,1] + -38.078;
   1:  PR[91,2] = PR[90,2] + -0.950;
   1:L PR[91] R[100]mm/sec CNT100;
   1:  PR[91,1] = PR[90,1] + -37.863;
   1:  PR[91,2] = PR[90,2] + -3.685;
   1:L PR[91] R[100]mm/sec CNT100;
   1:  PR[91,1] = PR[90,1] + -37.192;
   1:  PR[91,2] = PR[90,2] + -6.281;
   1:L PR[91] R[100]mm/sec CNT100;
   1:  PR[91,1] = PR[90,1] + -37.022;
   1:  PR[91,2] = PR[90,2] + -6.705;
   1:L PR[91] R[100]mm/sec CNT100;
   1:  PR[91,1] = PR[90,1] + -35.803;
   1:  PR[91,2] = PR[90,2] + -9.440;
   1:L PR[91] R[100]mm/sec CNT100;
   1:  PR[91,1] = PR[90,1] + -35.699;
   1:  PR[91,2] = PR[90,2] + -9.584;
   1:L PR[91] R[100]mm/sec CNT100;
   1:  PR[91,1] = PR[90,1] + -33.995;
   1:  PR[91,2] = PR[90,2] + -12.198;
   1:L PR[91] R[100]mm/sec CNT100;
   1:  PR[91,1] = PR[90,1] + -31.785;
   1:  PR[91,2] = PR[90,2] + -14.589;
   1:L PR[91] R[100]mm/sec CNT100;
   1:  PR[91,1] = PR[90,1] + -29.358;
   1:  PR[91,2] = PR[90,2] + -16.489;
   1:L PR[91] R[100]mm/sec CNT100;
   1:  PR[91,1] = PR[90,1] + -28.995;
   1:  PR[91,2] = PR[90,2] + -16.752;
   1:L PR[91] R[100]mm/sec CNT100;
   1:  PR[91,1] = PR[90,1] + -26.370;
   1:  PR[91,2] = PR[90,2] + -18.223;
   1:L PR[91] R[100]mm/sec CNT100;
   1:  PR[91,1] = PR[90,1] + -23.758;
   1:  PR[91,2] = PR[90,2] + -19.187;
   1:L PR[91] R[100]mm/sec CNT100;
   1:  PR[91,1] = PR[90,1] + -22.778;
   1:  PR[91,2] = PR[90,2] + -19.570;
   1:L PR[91] R[100]mm/sec CNT100;
   1:  PR[91,1] = PR[90,1] + -20.216;
   1:  PR[91,2] = PR[90,2] + -20.101;
   1:L PR[91] R[100]mm/sec CNT100;
   1:  PR[91,1] = PR[90,1] + -18.779;
   1:  PR[91,2] = PR[90,2] + -20.269;
   1:L PR[91] R[100]mm/sec CNT100;
   1:  PR[91,1] = PR[90,1] + -16.238;
   1:  PR[91,2] = PR[90,2] + -20.403;
   1:L PR[91] R[100]mm/sec CNT100;
   1:  PR[91,1] = PR[90,1] + -13.980;
   1:  PR[91,2] = PR[90,2] + -20.175;
   1:L PR[91] R[100]mm/sec CNT100;
   1:  PR[91,1] = PR[90,1] + -11.971;
   1:  PR[91,2] = PR[90,2] + -19.894;
   1:L PR[91] R[100]mm/sec CNT100;
   1:  PR[91,1] = PR[90,1] + -9.947;
   1:  PR[91,2] = PR[90,2] + -19.371;
   1:L PR[91] R[100]mm/sec CNT100;
   1:  PR[91,1] = PR[90,1] + -8.151;
   1:  PR[91,2] = PR[90,2] + -18.583;
   1:L PR[91] R[100]mm/sec CNT100;
   1:  PR[91,1] = PR[90,1] + -5.782;
   1:  PR[91,2] = PR[90,2] + -17.573;
   1:L PR[91] R[100]mm/sec CNT100;
   1:  PR[91,1] = PR[90,1] + -4.312;
   1:  PR[91,2] = PR[90,2] + -16.634;
   1:L PR[91] R[100]mm/sec CNT100;
   1:  PR[91,1] = PR[90,1] + -3.619;
   1:  PR[91,2] = PR[90,2] + -16.134;
   1:L PR[91] R[100]mm/sec CNT100;
   1:  PR[91,1] = PR[90,1] + -1.756;
   1:  PR[91,2] = PR[90,2] + -14.503;
   1:L PR[91] R[100]mm/sec CNT100;
   1:  PR[91,1] = PR[90,1] + -1.505;
   1:  PR[91,2] = PR[90,2] + -14.417;
   1:L PR[91] R[100]mm/sec CNT100;
   1:  PR[91,1] = PR[90,1] + -1.291;
   1:  PR[91,2] = PR[90,2] + -14.246;
   1:L PR[91] R[100]mm/sec CNT100;
   1:  PR[91,1] = PR[90,1] + -0.380;
   1:  PR[91,2] = PR[90,2] + -13.601;
   1:L PR[91] R[100]mm/sec CNT100;
   1:  PR[91,1] = PR[90,1] + 1.422;
   1:  PR[91,2] = PR[90,2] + -14.238;
   1:L PR[91] R[100]mm/sec CNT100;
   1:  PR[91,1] = PR[90,1] + 2.035;
   1:  PR[91,2] = PR[90,2] + -14.610;
   1:L PR[91] R[100]mm/sec CNT100;
   1:  PR[91,1] = PR[90,1] + 3.752;
   1:  PR[91,2] = PR[90,2] + -16.116;
   1:L PR[91] R[100]mm/sec CNT100;
   1:  PR[91,1] = PR[90,1] + 4.817;
   1:  PR[91,2] = PR[90,2] + -16.798;
   1:L PR[91] R[100]mm/sec CNT100;
   1:  PR[91,1] = PR[90,1] + 5.963;
   1:  PR[91,2] = PR[90,2] + -17.587;
   1:L PR[91] R[100]mm/sec CNT100;
   1:  PR[91,1] = PR[90,1] + 7.771;
   1:  PR[91,2] = PR[90,2] + -18.377;
   1:L PR[91] R[100]mm/sec CNT100;
   1:  PR[91,1] = PR[90,1] + 10.090;
   1:  PR[91,2] = PR[90,2] + -19.365;
   1:L PR[91] R[100]mm/sec CNT100;
   1:  PR[91,1] = PR[90,1] + 12.101;
   1:  PR[91,2] = PR[90,2] + -19.886;
   1:L PR[91] R[100]mm/sec CNT100;
   1:  PR[91,1] = PR[90,1] + 14.567;
   1:  PR[91,2] = PR[90,2] + -20.145;
   1:L PR[91] R[100]mm/sec CNT100;
   1:  PR[91,1] = PR[90,1] + 16.414;
   1:  PR[91,2] = PR[90,2] + -20.401;
   1:L PR[91] R[100]mm/sec CNT100;
   1:  PR[91,1] = PR[90,1] + 18.916;
   1:  PR[91,2] = PR[90,2] + -20.272;
   1:L PR[91] R[100]mm/sec CNT100;
   1:  PR[91,1] = PR[90,1] + 20.354;
   1:  PR[91,2] = PR[90,2] + -20.104;
   1:L PR[91] R[100]mm/sec CNT100;
   1:  PR[91,1] = PR[90,1] + 22.923;
   1:  PR[91,2] = PR[90,2] + -19.572;
   1:L PR[91] R[100]mm/sec CNT100;
   1:  PR[91,1] = PR[90,1] + 25.749;
   1:  PR[91,2] = PR[90,2] + -18.528;
   1:L PR[91] R[100]mm/sec CNT100;
   1:  PR[91,1] = PR[90,1] + 26.499;
   1:  PR[91,2] = PR[90,2] + -18.236;
   1:L PR[91] R[100]mm/sec CNT100;
   1:  PR[91,1] = PR[90,1] + 29.104;
   1:  PR[91,2] = PR[90,2] + -16.785;
   1:L PR[91] R[100]mm/sec CNT100;
   1:  PR[91,1] = PR[90,1] + 31.898;
   1:  PR[91,2] = PR[90,2] + -14.631;
   1:L PR[91] R[100]mm/sec CNT100;
   1:  PR[91,1] = PR[90,1] + 34.116;
   1:  PR[91,2] = PR[90,2] + -12.234;
   1:L PR[91] R[100]mm/sec CNT100;
   1:  PR[91,1] = PR[90,1] + 35.935;
   1:  PR[91,2] = PR[90,2] + -9.483;
   1:L PR[91] R[100]mm/sec CNT100;
   1:  PR[91,1] = PR[90,1] + 37.166;
   1:  PR[91,2] = PR[90,2] + -6.758;
   1:L PR[91] R[100]mm/sec CNT100;
   1:  PR[91,1] = PR[90,1] + 37.334;
   1:  PR[91,2] = PR[90,2] + -6.340;
   1:L PR[91] R[100]mm/sec CNT100;
   1:  PR[91,1] = PR[90,1] + 38.017;
   1:  PR[91,2] = PR[90,2] + -3.738;
   1:L PR[91] R[100]mm/sec CNT100;
   1:  PR[91,1] = PR[90,1] + 38.097;
   1:  PR[91,2] = PR[90,2] + -3.101;
   1:L PR[91] R[100]mm/sec CNT100;
   1:  PR[91,1] = PR[90,1] + 38.320;
   1:  PR[91,2] = PR[90,2] + -0.345;
   1:L PR[91] R[100]mm/sec CNT100;
   1:  PR[91,1] = PR[90,1] + 38.235;
   1:  PR[91,2] = PR[90,2] + 0.328;
   1:L PR[91] R[100]mm/sec CNT100;
   1:  PR[91,1] = PR[90,1] + 38.008;
   1:  PR[91,2] = PR[90,2] + 3.146;
   1:L PR[91] R[100]mm/sec CNT100;
   1:  PR[91,1] = PR[90,1] + 37.334;
   1:  PR[91,2] = PR[90,2] + 5.717;
   1:L PR[91] R[100]mm/sec CNT100;
   1:  PR[91,1] = PR[90,1] + 37.165;
   1:  PR[91,2] = PR[90,2] + 6.134;
   1:L PR[91] R[100]mm/sec CNT100;
   1:  PR[91,1] = PR[90,1] + 35.947;
   1:  PR[91,2] = PR[90,2] + 8.833;
   1:L PR[91] R[100]mm/sec CNT100;
   1:  PR[91,1] = PR[90,1] + 35.844;
   1:  PR[91,2] = PR[90,2] + 8.976;
   1:L PR[91] R[100]mm/sec CNT100;
   1:  PR[91,1] = PR[90,1] + 34.115;
   1:  PR[91,2] = PR[90,2] + 11.612;
   1:L PR[91] R[100]mm/sec CNT100;
   1:  PR[91,1] = PR[90,1] + 31.896;
   1:  PR[91,2] = PR[90,2] + 14.009;
   1:L PR[91] R[100]mm/sec CNT100;
   1:  PR[91,1] = PR[90,1] + 29.489;
   1:  PR[91,2] = PR[90,2] + 15.885;
   1:L PR[91] R[100]mm/sec CNT100;
   1:  PR[91,1] = PR[90,1] + 29.124;
   1:  PR[91,2] = PR[90,2] + 16.150;
   1:L PR[91] R[100]mm/sec CNT100;
   1:  PR[91,1] = PR[90,1] + 26.515;
   1:  PR[91,2] = PR[90,2] + 17.604;
   1:L PR[91] R[100]mm/sec CNT100;
   1:  PR[91,1] = PR[90,1] + 23.898;
   1:  PR[91,2] = PR[90,2] + 18.565;
   1:L PR[91] R[100]mm/sec CNT100;
   1:  PR[91,1] = PR[90,1] + 22.917;
   1:  PR[91,2] = PR[90,2] + 18.949;
   1:L PR[91] R[100]mm/sec CNT100;
   1:  PR[91,1] = PR[90,1] + 20.361;
   1:  PR[91,2] = PR[90,2] + 19.478;
   1:L PR[91] R[100]mm/sec CNT100;
   1:  PR[91,1] = PR[90,1] + 18.927;
   1:  PR[91,2] = PR[90,2] + 19.648;
   1:L PR[91] R[100]mm/sec CNT100;
   1:  PR[91,1] = PR[90,1] + 16.401;
   1:  PR[91,2] = PR[90,2] + 19.779;
   1:L PR[91] R[100]mm/sec CNT100;
   1:  PR[91,1] = PR[90,1] + 14.148;
   1:  PR[91,2] = PR[90,2] + 19.550;
   1:L PR[91] R[100]mm/sec CNT100;
   1:  PR[91,1] = PR[90,1] + 12.143;
   1:  PR[91,2] = PR[90,2] + 19.273;
   1:L PR[91] R[100]mm/sec CNT100;
   1:  PR[91,1] = PR[90,1] + 10.117;
   1:  PR[91,2] = PR[90,2] + 18.748;
   1:L PR[91] R[100]mm/sec CNT100;
   1:  PR[91,1] = PR[90,1] + 8.321;
   1:  PR[91,2] = PR[90,2] + 17.962;
   1:L PR[91] R[100]mm/sec CNT100;
   1:  PR[91,1] = PR[90,1] + 6.001;
   1:  PR[91,2] = PR[90,2] + 16.993;
   1:L PR[91] R[100]mm/sec CNT100;
   1:  PR[91,1] = PR[90,1] + 4.512;
   1:  PR[91,2] = PR[90,2] + 16.042;
   1:L PR[91] R[100]mm/sec CNT100;
   1:  PR[91,1] = PR[90,1] + 4.067;
   1:  PR[91,2] = PR[90,2] + 15.735;
   1:L PR[91] R[100]mm/sec CNT100;
   1:  PR[91,1] = PR[90,1] + 3.250;
   1:  PR[91,2] = PR[90,2] + 15.089;
   1:L PR[91] R[100]mm/sec CNT100;
   1:  PR[91,1] = PR[90,1] + 2.066;
   1:  PR[91,2] = PR[90,2] + 14.039;
   1:L PR[91] R[100]mm/sec CNT100;
   1:  PR[91,1] = PR[90,1] + 1.546;
   1:  PR[91,2] = PR[90,2] + 13.686;
   1:L PR[91] R[100]mm/sec CNT100;
   1:  PR[91,1] = PR[90,1] + 0.531;
   1:  PR[91,2] = PR[90,2] + 13.144;
   1:L PR[91] R[100]mm/sec CNT100;
   1:  PR[91,1] = PR[90,1] + -0.464;
   1:L PR[91] R[100]mm/sec CNT100;
   1:  PR[91] = PR[90];
   1:  PR[91,1] = PR[90,1] + -1.737;
   1:  PR[91,2] = PR[90,2] + 14.036;
   1:  PR[91,3] = PR[90,3] + 31.415;
   1:L PR[91] R[100]mm/sec CNT100;
   1:  PR[91,1] = PR[90,1] + -2.061;
   1:  PR[91,2] = PR[90,2] + 14.458;
   1:L PR[91] R[100]mm/sec CNT100;
   1:  PR[91,1] = PR[90,1] + -2.803;
   1:  PR[91,2] = PR[90,2] + 15.114;
   1:L PR[91] R[100]mm/sec CNT100;
   1:  PR[91,1] = PR[90,1] + -3.663;
   1:  PR[91,2] = PR[90,2] + 15.794;
   1:L PR[91] R[100]mm/sec CNT100;
   1:  PR[91,1] = PR[90,1] + -4.821;
   1:  PR[91,2] = PR[90,2] + 16.536;
   1:L PR[91] R[100]mm/sec CNT100;
   1:  PR[91,1] = PR[90,1] + -5.585;
   1:  PR[91,2] = PR[90,2] + 17.048;
   1:L PR[91] R[100]mm/sec CNT100;
   1:  PR[91,1] = PR[90,1] + -7.301;
   1:  PR[91,2] = PR[90,2] + 17.798;
   1:L PR[91] R[100]mm/sec CNT100;
   1:  PR[91,1] = PR[90,1] + -9.760;
   1:  PR[91,2] = PR[90,2] + 18.828;
   1:L PR[91] R[100]mm/sec CNT100;
   1:  PR[91,1] = PR[90,1] + -11.641;
   1:  PR[91,2] = PR[90,2] + 19.314;
   1:L PR[91] R[100]mm/sec CNT100;
   1:  PR[91,1] = PR[90,1] + -13.962;
   1:  PR[91,2] = PR[90,2] + 19.556;
   1:L PR[91] R[100]mm/sec CNT100;
   1:  PR[91,1] = PR[90,1] + -16.053;
   1:  PR[91,2] = PR[90,2] + 19.841;
   1:L PR[91] R[100]mm/sec CNT100;
   1:  PR[91,1] = PR[90,1] + -18.424;
   1:  PR[91,2] = PR[90,2] + 19.716;
   1:L PR[91] R[100]mm/sec CNT100;
   1:  PR[91,1] = PR[90,1] + -20.099;
   1:  PR[91,2] = PR[90,2] + 19.518;
   1:L PR[91] R[100]mm/sec CNT100;
   1:  PR[91,1] = PR[90,1] + -22.538;
   1:  PR[91,2] = PR[90,2] + 19.012;
   1:L PR[91] R[100]mm/sec CNT100;
   1:  PR[91,1] = PR[90,1] + -25.216;
   1:  PR[91,2] = PR[90,2] + 18.018;
   1:L PR[91] R[100]mm/sec CNT100;
   1:  PR[91,1] = PR[90,1] + -26.201;
   1:  PR[91,2] = PR[90,2] + 17.633;
   1:L PR[91] R[100]mm/sec CNT100;
   1:  PR[91,1] = PR[90,1] + -28.688;
   1:  PR[91,2] = PR[90,2] + 16.240;
   1:L PR[91] R[100]mm/sec CNT100;
   1:  PR[91,1] = PR[90,1] + -31.245;
   1:  PR[91,2] = PR[90,2] + 14.250;
   1:L PR[91] R[100]mm/sec CNT100;
   1:  PR[91,1] = PR[90,1] + -31.607;
   1:  PR[91,2] = PR[90,2] + 13.986;
   1:L PR[91] R[100]mm/sec CNT100;
   1:  PR[91,1] = PR[90,1] + -33.725;
   1:  PR[91,2] = PR[90,2] + 11.698;
   1:L PR[91] R[100]mm/sec CNT100;
   1:  PR[91,1] = PR[90,1] + -33.835;
   1:  PR[91,2] = PR[90,2] + 11.562;
   1:L PR[91] R[100]mm/sec CNT100;
   1:  PR[91,1] = PR[90,1] + -35.600;
   1:  PR[91,2] = PR[90,2] + 8.880;
   1:L PR[91] R[100]mm/sec CNT100;
   1:  PR[91,1] = PR[90,1] + -36.981;
   1:  PR[91,2] = PR[90,2] + 5.781;
   1:L PR[91] R[100]mm/sec CNT100;
   1:  PR[91,1] = PR[90,1] + -37.733;
   1:  PR[91,2] = PR[90,2] + 2.874;
   1:L PR[91] R[100]mm/sec CNT100;
   1:  PR[91,1] = PR[90,1] + -37.753;
   1:  PR[91,2] = PR[90,2] + 2.713;
   1:L PR[91] R[100]mm/sec CNT100;
   1:  PR[91,1] = PR[90,1] + -37.990;
   1:  PR[91,2] = PR[90,2] + -0.277;
   1:L PR[91] R[100]mm/sec CNT100;
   1:  PR[91,1] = PR[90,1] + -37.963;
   1:  PR[91,2] = PR[90,2] + -0.490;
   1:L PR[91] R[100]mm/sec CNT100;
   1:  PR[91,1] = PR[90,1] + -37.724;
   1:  PR[91,2] = PR[90,2] + -3.531;
   1:L PR[91] R[100]mm/sec CNT100;
   1:  PR[91,1] = PR[90,1] + -36.981;
   1:  PR[91,2] = PR[90,2] + -6.405;
   1:L PR[91] R[100]mm/sec CNT100;
   1:  PR[91,1] = PR[90,1] + -35.600;
   1:  PR[91,2] = PR[90,2] + -9.504;
   1:L PR[91] R[100]mm/sec CNT100;
   1:  PR[91,1] = PR[90,1] + -33.835;
   1:  PR[91,2] = PR[90,2] + -12.186;
   1:L PR[91] R[100]mm/sec CNT100;
   1:  PR[91,1] = PR[90,1] + -33.725;
   1:  PR[91,2] = PR[90,2] + -12.322;
   1:L PR[91] R[100]mm/sec CNT100;
   1:  PR[91,1] = PR[90,1] + -31.589;
   1:  PR[91,2] = PR[90,2] + -14.630;
   1:L PR[91] R[100]mm/sec CNT100;
   1:  PR[91,1] = PR[90,1] + -29.269;
   1:  PR[91,2] = PR[90,2] + -16.445;
   1:L PR[91] R[100]mm/sec CNT100;
   1:  PR[91,1] = PR[90,1] + -28.706;
   1:  PR[91,2] = PR[90,2] + -16.854;
   1:L PR[91] R[100]mm/sec CNT100;
   1:  PR[91,1] = PR[90,1] + -26.208;
   1:  PR[91,2] = PR[90,2] + -18.253;
   1:L PR[91] R[100]mm/sec CNT100;
   1:  PR[91,1] = PR[90,1] + -23.718;
   1:  PR[91,2] = PR[90,2] + -19.173;
   1:L PR[91] R[100]mm/sec CNT100;
   1:  PR[91,1] = PR[90,1] + -22.518;
   1:  PR[91,2] = PR[90,2] + -19.641;
   1:L PR[91] R[100]mm/sec CNT100;
   1:  PR[91,1] = PR[90,1] + -20.089;
   1:  PR[91,2] = PR[90,2] + -20.145;
   1:L PR[91] R[100]mm/sec CNT100;
   1:  PR[91,1] = PR[90,1] + -18.410;
   1:  PR[91,2] = PR[90,2] + -20.340;
   1:L PR[91] R[100]mm/sec CNT100;
   1:  PR[91,1] = PR[90,1] + -16.012;
   1:  PR[91,2] = PR[90,2] + -20.467;
   1:L PR[91] R[100]mm/sec CNT100;
   1:  PR[91,1] = PR[90,1] + -13.881;
   1:  PR[91,2] = PR[90,2] + -20.252;
   1:L PR[91] R[100]mm/sec CNT100;
   1:  PR[91,1] = PR[90,1] + -11.644;
   1:  PR[91,2] = PR[90,2] + -19.939;
   1:L PR[91] R[100]mm/sec CNT100;
   1:  PR[91,1] = PR[90,1] + -9.749;
   1:  PR[91,2] = PR[90,2] + -19.449;
   1:L PR[91] R[100]mm/sec CNT100;
   1:  PR[91,1] = PR[90,1] + -8.064;
   1:  PR[91,2] = PR[90,2] + -18.710;
   1:L PR[91] R[100]mm/sec CNT100;
   1:  PR[91,1] = PR[90,1] + -5.488;
   1:  PR[91,2] = PR[90,2] + -17.612;
   1:L PR[91] R[100]mm/sec CNT100;
   1:  PR[91,1] = PR[90,1] + -4.127;
   1:  PR[91,2] = PR[90,2] + -16.742;
   1:L PR[91] R[100]mm/sec CNT100;
   1:  PR[91,1] = PR[90,1] + -3.375;
   1:  PR[91,2] = PR[90,2] + -16.200;
   1:L PR[91] R[100]mm/sec CNT100;
   1:  PR[91,1] = PR[90,1] + -1.738;
   1:  PR[91,2] = PR[90,2] + -14.767;
   1:L PR[91] R[100]mm/sec CNT100;
   1:  PR[91,1] = PR[90,1] + -1.337;
   1:  PR[91,2] = PR[90,2] + -14.630;
   1:L PR[91] R[100]mm/sec CNT100;
   1:  PR[91,1] = PR[90,1] + -0.386;
   1:  PR[91,2] = PR[90,2] + -13.904;
   1:L PR[91] R[100]mm/sec CNT100;
   1:  PR[91,1] = PR[90,1] + 0.996;
   1:  PR[91,2] = PR[90,2] + -14.395;
   1:L PR[91] R[100]mm/sec CNT100;
   1:  PR[91,1] = PR[90,1] + 1.349;
   1:  PR[91,2] = PR[90,2] + -14.458;
   1:L PR[91] R[100]mm/sec CNT100;
   1:  PR[91,1] = PR[90,1] + 2.023;
   1:  PR[91,2] = PR[90,2] + -14.880;
   1:L PR[91] R[100]mm/sec CNT100;
   1:  PR[91,1] = PR[90,1] + 3.507;
   1:  PR[91,2] = PR[90,2] + -16.181;
   1:L PR[91] R[100]mm/sec CNT100;
   1:  PR[91,1] = PR[90,1] + 4.420;
   1:  PR[91,2] = PR[90,2] + -16.766;
   1:L PR[91] R[100]mm/sec CNT100;
   1:  PR[91,1] = PR[90,1] + 5.669;
   1:  PR[91,2] = PR[90,2] + -17.626;
   1:L PR[91] R[100]mm/sec CNT100;
   1:  PR[91,1] = PR[90,1] + 7.347;
   1:  PR[91,2] = PR[90,2] + -18.359;
   1:L PR[91] R[100]mm/sec CNT100;
   1:  PR[91,1] = PR[90,1] + 9.893;
   1:  PR[91,2] = PR[90,2] + -19.443;
   1:L PR[91] R[100]mm/sec CNT100;
   1:  PR[91,1] = PR[90,1] + 11.774;
   1:  PR[91,2] = PR[90,2] + -19.931;
   1:L PR[91] R[100]mm/sec CNT100;
   1:  PR[91,1] = PR[90,1] + 14.091;
   1:  PR[91,2] = PR[90,2] + -20.174;
   1:L PR[91] R[100]mm/sec CNT100;
   1:  PR[91,1] = PR[90,1] + 16.188;
   1:  PR[91,2] = PR[90,2] + -20.465;
   1:L PR[91] R[100]mm/sec CNT100;
   1:  PR[91,1] = PR[90,1] + 18.547;
   1:  PR[91,2] = PR[90,2] + -20.343;
   1:L PR[91] R[100]mm/sec CNT100;
   1:  PR[91,1] = PR[90,1] + 20.228;
   1:  PR[91,2] = PR[90,2] + -20.147;
   1:L PR[91] R[100]mm/sec CNT100;
   1:  PR[91,1] = PR[90,1] + 22.665;
   1:  PR[91,2] = PR[90,2] + -19.643;
   1:L PR[91] R[100]mm/sec CNT100;
   1:  PR[91,1] = PR[90,1] + 25.348;
   1:  PR[91,2] = PR[90,2] + -18.652;
   1:L PR[91] R[100]mm/sec CNT100;
   1:  PR[91,1] = PR[90,1] + 26.337;
   1:  PR[91,2] = PR[90,2] + -18.267;
   1:L PR[91] R[100]mm/sec CNT100;
   1:  PR[91,1] = PR[90,1] + 28.815;
   1:  PR[91,2] = PR[90,2] + -16.886;
   1:L PR[91] R[100]mm/sec CNT100;
   1:  PR[91,1] = PR[90,1] + 31.351;
   1:  PR[91,2] = PR[90,2] + -14.921;
   1:L PR[91] R[100]mm/sec CNT100;
   1:  PR[91,1] = PR[90,1] + 31.718;
   1:  PR[91,2] = PR[90,2] + -14.655;
   1:L PR[91] R[100]mm/sec CNT100;
   1:  PR[91,1] = PR[90,1] + 33.841;
   1:  PR[91,2] = PR[90,2] + -12.364;
   1:L PR[91] R[100]mm/sec CNT100;
   1:  PR[91,1] = PR[90,1] + 33.955;
   1:  PR[91,2] = PR[90,2] + -12.223;
   1:L PR[91] R[100]mm/sec CNT100;
   1:  PR[91,1] = PR[90,1] + 35.744;
   1:  PR[91,2] = PR[90,2] + -9.519;
   1:L PR[91] R[100]mm/sec CNT100;
   1:  PR[91,1] = PR[90,1] + 36.572;
   1:  PR[91,2] = PR[90,2] + -7.697;
   1:L PR[91] R[100]mm/sec CNT100;
   1:  PR[91,1] = PR[90,1] + 37.122;
   1:  PR[91,2] = PR[90,2] + -6.469;
   1:L PR[91] R[100]mm/sec CNT100;
   1:  PR[91,1] = PR[90,1] + 37.876;
   1:  PR[91,2] = PR[90,2] + -3.591;
   1:L PR[91] R[100]mm/sec CNT100;
   1:  PR[91,1] = PR[90,1] + 37.896;
   1:  PR[91,2] = PR[90,2] + -3.433;
   1:L PR[91] R[100]mm/sec CNT100;
   1:  PR[91,1] = PR[90,1] + 38.147;
   1:  PR[91,2] = PR[90,2] + -0.345;
   1:L PR[91] R[100]mm/sec CNT100;
   1:  PR[91,1] = PR[90,1] + 38.120;
   1:  PR[91,2] = PR[90,2] + -0.134;
   1:L PR[91] R[100]mm/sec CNT100;
   1:  PR[91,1] = PR[90,1] + 37.868;
   1:  PR[91,2] = PR[90,2] + 2.999;
   1:L PR[91] R[100]mm/sec CNT100;
   1:  PR[91,1] = PR[90,1] + 37.122;
   1:  PR[91,2] = PR[90,2] + 5.843;
   1:L PR[91] R[100]mm/sec CNT100;
   1:  PR[91,1] = PR[90,1] + 35.744;
   1:  PR[91,2] = PR[90,2] + 8.896;
   1:L PR[91] R[100]mm/sec CNT100;
   1:  PR[91,1] = PR[90,1] + 33.955;
   1:  PR[91,2] = PR[90,2] + 11.599;
   1:L PR[91] R[100]mm/sec CNT100;
   1:  PR[91,1] = PR[90,1] + 33.842;
   1:  PR[91,2] = PR[90,2] + 11.740;
   1:L PR[91] R[100]mm/sec CNT100;
   1:  PR[91,1] = PR[90,1] + 31.702;
   1:  PR[91,2] = PR[90,2] + 14.047;
   1:L PR[91] R[100]mm/sec CNT100;
   1:  PR[91,1] = PR[90,1] + 29.402;
   1:  PR[91,2] = PR[90,2] + 15.840;
   1:L PR[91] R[100]mm/sec CNT100;
   1:  PR[91,1] = PR[90,1] + 28.838;
   1:  PR[91,2] = PR[90,2] + 16.249;
   1:L PR[91] R[100]mm/sec CNT100;
   1:  PR[91,1] = PR[90,1] + 26.354;
   1:  PR[91,2] = PR[90,2] + 17.634;
   1:L PR[91] R[100]mm/sec CNT100;
   1:  PR[91,1] = PR[90,1] + 23.860;
   1:  PR[91,2] = PR[90,2] + 18.550;
   1:L PR[91] R[100]mm/sec CNT100;
   1:  PR[91,1] = PR[90,1] + 22.660;
   1:  PR[91,2] = PR[90,2] + 19.019;
   1:L PR[91] R[100]mm/sec CNT100;
   1:  PR[91,1] = PR[90,1] + 20.237;
   1:  PR[91,2] = PR[90,2] + 19.521;
   1:L PR[91] R[100]mm/sec CNT100;
   1:  PR[91,1] = PR[90,1] + 18.561;
   1:  PR[91,2] = PR[90,2] + 19.719;
   1:L PR[91] R[100]mm/sec CNT100;
   1:  PR[91,1] = PR[90,1] + 16.177;
   1:  PR[91,2] = PR[90,2] + 19.843;
   1:L PR[91] R[100]mm/sec CNT100;
   1:  PR[91,1] = PR[90,1] + 14.051;
   1:  PR[91,2] = PR[90,2] + 19.627;
   1:L PR[91] R[100]mm/sec CNT100;
   1:  PR[91,1] = PR[90,1] + 11.818;
   1:  PR[91,2] = PR[90,2] + 19.319;
   1:L PR[91] R[100]mm/sec CNT100;
   1:  PR[91,1] = PR[90,1] + 9.921;
   1:  PR[91,2] = PR[90,2] + 18.827;
   1:L PR[91] R[100]mm/sec CNT100;
   1:  PR[91,1] = PR[90,1] + 8.235;
   1:  PR[91,2] = PR[90,2] + 18.089;
   1:L PR[91] R[100]mm/sec CNT100;
   1:  PR[91,1] = PR[90,1] + 5.713;
   1:  PR[91,2] = PR[90,2] + 17.035;
   1:L PR[91] R[100]mm/sec CNT100;
   1:  PR[91,1] = PR[90,1] + 4.329;
   1:  PR[91,2] = PR[90,2] + 16.152;
   1:L PR[91] R[100]mm/sec CNT100;
   1:  PR[91,1] = PR[90,1] + 3.846;
   1:  PR[91,2] = PR[90,2] + 15.818;
   1:L PR[91] R[100]mm/sec CNT100;
   1:  PR[91,1] = PR[90,1] + 2.962;
   1:  PR[91,2] = PR[90,2] + 15.119;
   1:L PR[91] R[100]mm/sec CNT100;
   1:  PR[91,1] = PR[90,1] + 2.045;
   1:  PR[91,2] = PR[90,2] + 14.306;
   1:L PR[91] R[100]mm/sec CNT100;
   1:  PR[91,1] = PR[90,1] + 1.786;
   1:  PR[91,2] = PR[90,2] + 14.131;
   1:L PR[91] R[100]mm/sec CNT100;
   1:  PR[91,1] = PR[90,1] + 1.502;
   1:  PR[91,2] = PR[90,2] + 13.855;
   1:L PR[91] R[100]mm/sec CNT100;
   1:  PR[91,1] = PR[90,1] + 1.098;
   1:  PR[91,2] = PR[90,2] + 13.786;
   1:L PR[91] R[100]mm/sec CNT100;
   1:  PR[91,1] = PR[90,1] + 0.499;
   1:  PR[91,2] = PR[90,2] + 13.458;
   1:L PR[91] R[100]mm/sec CNT100;
   1:  PR[91,1] = PR[90,1] + -0.440;
   1:L PR[91] R[100]mm/sec CNT100;
   1:  PR[91] = PR[90];
   1:  PR[91,1] = PR[90,1] + -1.776;
   1:  PR[91,2] = PR[90,2] + 14.379;
   1:  PR[91,3] = PR[90,3] + 32.025;
   1:L PR[91] R[100]mm/sec CNT100;
   1:  PR[91,1] = PR[90,1] + -2.043;
   1:  PR[91,2] = PR[90,2] + 14.727;
   1:L PR[91] R[100]mm/sec CNT100;
   1:  PR[91,1] = PR[90,1] + -2.516;
   1:  PR[91,2] = PR[90,2] + 15.145;
   1:L PR[91] R[100]mm/sec CNT100;
   1:  PR[91,1] = PR[90,1] + -3.443;
   1:  PR[91,2] = PR[90,2] + 15.878;
   1:L PR[91] R[100]mm/sec CNT100;
   1:  PR[91,1] = PR[90,1] + -4.468;
   1:  PR[91,2] = PR[90,2] + 16.534;
   1:L PR[91] R[100]mm/sec CNT100;
   1:  PR[91,1] = PR[90,1] + -5.298;
   1:  PR[91,2] = PR[90,2] + 17.091;
   1:L PR[91] R[100]mm/sec CNT100;
   1:  PR[91,1] = PR[90,1] + -6.886;
   1:  PR[91,2] = PR[90,2] + 17.785;
   1:L PR[91] R[100]mm/sec CNT100;
   1:  PR[91,1] = PR[90,1] + -9.564;
   1:  PR[91,2] = PR[90,2] + 18.907;
   1:L PR[91] R[100]mm/sec CNT100;
   1:  PR[91,1] = PR[90,1] + -11.316;
   1:  PR[91,2] = PR[90,2] + 19.360;
   1:L PR[91] R[100]mm/sec CNT100;
   1:  PR[91,1] = PR[90,1] + -13.488;
   1:  PR[91,2] = PR[90,2] + 19.586;
   1:L PR[91] R[100]mm/sec CNT100;
   1:  PR[91,1] = PR[90,1] + -15.829;
   1:  PR[91,2] = PR[90,2] + 19.905;
   1:L PR[91] R[100]mm/sec CNT100;
   1:  PR[91,1] = PR[90,1] + -18.057;
   1:  PR[91,2] = PR[90,2] + 19.788;
   1:L PR[91] R[100]mm/sec CNT100;
   1:  PR[91,1] = PR[90,1] + -19.974;
   1:  PR[91,2] = PR[90,2] + 19.561;
   1:L PR[91] R[100]mm/sec CNT100;
   1:  PR[91,1] = PR[90,1] + -22.280;
   1:  PR[91,2] = PR[90,2] + 19.083;
   1:L PR[91] R[100]mm/sec CNT100;
   1:  PR[91,1] = PR[90,1] + -24.815;
   1:  PR[91,2] = PR[90,2] + 18.142;
   1:L PR[91] R[100]mm/sec CNT100;
   1:  PR[91,1] = PR[90,1] + -26.039;
   1:  PR[91,2] = PR[90,2] + 17.663;
   1:L PR[91] R[100]mm/sec CNT100;
   1:  PR[91,1] = PR[90,1] + -28.400;
   1:  PR[91,2] = PR[90,2] + 16.340;
   1:L PR[91] R[100]mm/sec CNT100;
   1:  PR[91,1] = PR[90,1] + -30.833;
   1:  PR[91,2] = PR[90,2] + 14.447;
   1:L PR[91] R[100]mm/sec CNT100;
   1:  PR[91,1] = PR[90,1] + -31.411;
   1:  PR[91,2] = PR[90,2] + 14.026;
   1:L PR[91] R[100]mm/sec CNT100;
   1:  PR[91,1] = PR[90,1] + -33.429;
   1:  PR[91,2] = PR[90,2] + 11.846;
   1:L PR[91] R[100]mm/sec CNT100;
   1:  PR[91,1] = PR[90,1] + -33.699;
   1:  PR[91,2] = PR[90,2] + 11.511;
   1:L PR[91] R[100]mm/sec CNT100;
   1:  PR[91,1] = PR[90,1] + -35.386;
   1:  PR[91,2] = PR[90,2] + 8.948;
   1:L PR[91] R[100]mm/sec CNT100;
   1:  PR[91,1] = PR[90,1] + -36.796;
   1:  PR[91,2] = PR[90,2] + 5.798;
   1:L PR[91] R[100]mm/sec CNT100;
   1:  PR[91,1] = PR[90,1] + -37.557;
   1:  PR[91,2] = PR[90,2] + 2.858;
   1:L PR[91] R[100]mm/sec CNT100;
   1:  PR[91,1] = PR[90,1] + -37.815;
   1:  PR[91,2] = PR[90,2] + -0.313;
   1:L PR[91] R[100]mm/sec CNT100;
   1:  PR[91,1] = PR[90,1] + -37.566;
   1:  PR[91,2] = PR[90,2] + -3.449;
   1:L PR[91] R[100]mm/sec CNT100;
   1:  PR[91,1] = PR[90,1] + -36.796;
   1:  PR[91,2] = PR[90,2] + -6.422;
   1:L PR[91] R[100]mm/sec CNT100;
   1:  PR[91,1] = PR[90,1] + -35.470;
   1:  PR[91,2] = PR[90,2] + -9.377;
   1:L PR[91] R[100]mm/sec CNT100;
   1:  PR[91,1] = PR[90,1] + -35.382;
   1:  PR[91,2] = PR[90,2] + -9.577;
   1:L PR[91] R[100]mm/sec CNT100;
   1:  PR[91,1] = PR[90,1] + -33.699;
   1:  PR[91,2] = PR[90,2] + -12.135;
   1:L PR[91] R[100]mm/sec CNT100;
   1:  PR[91,1] = PR[90,1] + -33.428;
   1:  PR[91,2] = PR[90,2] + -12.471;
   1:L PR[91] R[100]mm/sec CNT100;
   1:  PR[91,1] = PR[90,1] + -31.392;
   1:  PR[91,2] = PR[90,2] + -14.670;
   1:L PR[91] R[100]mm/sec CNT100;
   1:  PR[91,1] = PR[90,1] + -29.180;
   1:  PR[91,2] = PR[90,2] + -16.402;
   1:L PR[91] R[100]mm/sec CNT100;
   1:  PR[91,1] = PR[90,1] + -28.417;
   1:  PR[91,2] = PR[90,2] + -16.955;
   1:L PR[91] R[100]mm/sec CNT100;
   1:  PR[91,1] = PR[90,1] + -26.045;
   1:  PR[91,2] = PR[90,2] + -18.284;
   1:L PR[91] R[100]mm/sec CNT100;
   1:  PR[91,1] = PR[90,1] + -23.677;
   1:  PR[91,2] = PR[90,2] + -19.158;
   1:L PR[91] R[100]mm/sec CNT100;
   1:  PR[91,1] = PR[90,1] + -22.258;
   1:  PR[91,2] = PR[90,2] + -19.712;
   1:L PR[91] R[100]mm/sec CNT100;
   1:  PR[91,1] = PR[90,1] + -19.963;
   1:  PR[91,2] = PR[90,2] + -20.188;
   1:L PR[91] R[100]mm/sec CNT100;
   1:  PR[91,1] = PR[90,1] + -18.041;
   1:  PR[91,2] = PR[90,2] + -20.412;
   1:L PR[91] R[100]mm/sec CNT100;
   1:  PR[91,1] = PR[90,1] + -15.786;
   1:  PR[91,2] = PR[90,2] + -20.531;
   1:L PR[91] R[100]mm/sec CNT100;
   1:  PR[91,1] = PR[90,1] + -13.783;
   1:  PR[91,2] = PR[90,2] + -20.329;
   1:L PR[91] R[100]mm/sec CNT100;
   1:  PR[91,1] = PR[90,1] + -11.317;
   1:  PR[91,2] = PR[90,2] + -19.984;
   1:L PR[91] R[100]mm/sec CNT100;
   1:  PR[91,1] = PR[90,1] + -9.551;
   1:  PR[91,2] = PR[90,2] + -19.527;
   1:L PR[91] R[100]mm/sec CNT100;
   1:  PR[91,1] = PR[90,1] + -7.977;
   1:  PR[91,2] = PR[90,2] + -18.837;
   1:L PR[91] R[100]mm/sec CNT100;
   1:  PR[91,1] = PR[90,1] + -5.195;
   1:  PR[91,2] = PR[90,2] + -17.651;
   1:L PR[91] R[100]mm/sec CNT100;
   1:  PR[91,1] = PR[90,1] + -3.942;
   1:  PR[91,2] = PR[90,2] + -16.850;
   1:L PR[91] R[100]mm/sec CNT100;
   1:  PR[91,1] = PR[90,1] + -3.131;
   1:  PR[91,2] = PR[90,2] + -16.265;
   1:L PR[91] R[100]mm/sec CNT100;
   1:  PR[91,1] = PR[90,1] + -1.721;
   1:  PR[91,2] = PR[90,2] + -15.030;
   1:L PR[91] R[100]mm/sec CNT100;
   1:  PR[91,1] = PR[90,1] + -1.186;
   1:  PR[91,2] = PR[90,2] + -14.848;
   1:L PR[91] R[100]mm/sec CNT100;
   1:  PR[91,1] = PR[90,1] + -0.361;
   1:  PR[91,2] = PR[90,2] + -14.219;
   1:L PR[91] R[100]mm/sec CNT100;
   1:  PR[91,1] = PR[90,1] + 0.835;
   1:  PR[91,2] = PR[90,2] + -14.644;
   1:L PR[91] R[100]mm/sec CNT100;
   1:  PR[91,1] = PR[90,1] + 1.381;
   1:  PR[91,2] = PR[90,2] + -14.742;
   1:L PR[91] R[100]mm/sec CNT100;
   1:  PR[91,1] = PR[90,1] + 2.014;
   1:  PR[91,2] = PR[90,2] + -15.151;
   1:L PR[91] R[100]mm/sec CNT100;
   1:  PR[91,1] = PR[90,1] + 3.262;
   1:  PR[91,2] = PR[90,2] + -16.245;
   1:L PR[91] R[100]mm/sec CNT100;
   1:  PR[91,1] = PR[90,1] + 4.033;
   1:  PR[91,2] = PR[90,2] + -16.740;
   1:L PR[91] R[100]mm/sec CNT100;
   1:  PR[91,1] = PR[90,1] + 4.585;
   1:  PR[91,2] = PR[90,2] + -17.133;
   1:L PR[91] R[100]mm/sec CNT100;
   1:  PR[91,1] = PR[90,1] + 5.370;
   1:  PR[91,2] = PR[90,2] + -17.662;
   1:L PR[91] R[100]mm/sec CNT100;
   1:  PR[91,1] = PR[90,1] + 6.923;
   1:  PR[91,2] = PR[90,2] + -18.340;
   1:L PR[91] R[100]mm/sec CNT100;
   1:  PR[91,1] = PR[90,1] + 9.695;
   1:  PR[91,2] = PR[90,2] + -19.522;
   1:L PR[91] R[100]mm/sec CNT100;
   1:  PR[91,1] = PR[90,1] + 11.447;
   1:  PR[91,2] = PR[90,2] + -19.976;
   1:L PR[91] R[100]mm/sec CNT100;
   1:  PR[91,1] = PR[90,1] + 13.616;
   1:  PR[91,2] = PR[90,2] + -20.203;
   1:L PR[91] R[100]mm/sec CNT100;
   1:  PR[91,1] = PR[90,1] + 15.963;
   1:  PR[91,2] = PR[90,2] + -20.529;
   1:L PR[91] R[100]mm/sec CNT100;
   1:  PR[91,1] = PR[90,1] + 18.179;
   1:  PR[91,2] = PR[90,2] + -20.414;
   1:L PR[91] R[100]mm/sec CNT100;
   1:  PR[91,1] = PR[90,1] + 20.102;
   1:  PR[91,2] = PR[90,2] + -20.190;
   1:L PR[91] R[100]mm/sec CNT100;
   1:  PR[91,1] = PR[90,1] + 22.406;
   1:  PR[91,2] = PR[90,2] + -19.714;
   1:L PR[91] R[100]mm/sec CNT100;
   1:  PR[91,1] = PR[90,1] + 24.945;
   1:  PR[91,2] = PR[90,2] + -18.775;
   1:L PR[91] R[100]mm/sec CNT100;
   1:  PR[91,1] = PR[90,1] + 26.175;
   1:  PR[91,2] = PR[90,2] + -18.297;
   1:L PR[91] R[100]mm/sec CNT100;
   1:  PR[91,1] = PR[90,1] + 28.527;
   1:  PR[91,2] = PR[90,2] + -16.987;
   1:L PR[91] R[100]mm/sec CNT100;
   1:  PR[91,1] = PR[90,1] + 30.940;
   1:  PR[91,2] = PR[90,2] + -15.117;
   1:L PR[91] R[100]mm/sec CNT100;
   1:  PR[91,1] = PR[90,1] + 31.523;
   1:  PR[91,2] = PR[90,2] + -14.693;
   1:L PR[91] R[100]mm/sec CNT100;
   1:  PR[91,1] = PR[90,1] + 33.546;
   1:  PR[91,2] = PR[90,2] + -12.511;
   1:L PR[91] R[100]mm/sec CNT100;
   1:  PR[91,1] = PR[90,1] + 33.820;
   1:  PR[91,2] = PR[90,2] + -12.171;
   1:L PR[91] R[100]mm/sec CNT100;
   1:  PR[91,1] = PR[90,1] + 35.530;
   1:  PR[91,2] = PR[90,2] + -9.588;
   1:L PR[91] R[100]mm/sec CNT100;
   1:  PR[91,1] = PR[90,1] + 36.906;
   1:  PR[91,2] = PR[90,2] + -6.556;
   1:L PR[91] R[100]mm/sec CNT100;
   1:  PR[91,1] = PR[90,1] + 36.935;
   1:  PR[91,2] = PR[90,2] + -6.490;
   1:L PR[91] R[100]mm/sec CNT100;
   1:  PR[91,1] = PR[90,1] + 37.700;
   1:  PR[91,2] = PR[90,2] + -3.579;
   1:L PR[91] R[100]mm/sec CNT100;
   1:  PR[91,1] = PR[90,1] + 37.972;
   1:  PR[91,2] = PR[90,2] + -0.312;
   1:L PR[91] R[100]mm/sec CNT100;
   1:  PR[91,1] = PR[90,1] + 37.700;
   1:  PR[91,2] = PR[90,2] + 2.954;
   1:L PR[91] R[100]mm/sec CNT100;
   1:  PR[91,1] = PR[90,1] + 36.937;
   1:  PR[91,2] = PR[90,2] + 5.858;
   1:L PR[91] R[100]mm/sec CNT100;
   1:  PR[91,1] = PR[90,1] + 35.530;
   1:  PR[91,2] = PR[90,2] + 8.963;
   1:L PR[91] R[100]mm/sec CNT100;
   1:  PR[91,1] = PR[90,1] + 33.821;
   1:  PR[91,2] = PR[90,2] + 11.546;
   1:L PR[91] R[100]mm/sec CNT100;
   1:  PR[91,1] = PR[90,1] + 33.547;
   1:  PR[91,2] = PR[90,2] + 11.886;
   1:L PR[91] R[100]mm/sec CNT100;
   1:  PR[91,1] = PR[90,1] + 31.508;
   1:  PR[91,2] = PR[90,2] + 14.085;
   1:L PR[91] R[100]mm/sec CNT100;
   1:  PR[91,1] = PR[90,1] + 29.314;
   1:  PR[91,2] = PR[90,2] + 15.795;
   1:L PR[91] R[100]mm/sec CNT100;
   1:  PR[91,1] = PR[90,1] + 28.552;
   1:  PR[91,2] = PR[90,2] + 16.349;
   1:L PR[91] R[100]mm/sec CNT100;
   1:  PR[91,1] = PR[90,1] + 26.193;
   1:  PR[91,2] = PR[90,2] + 17.663;
   1:L PR[91] R[100]mm/sec CNT100;
   1:  PR[91,1] = PR[90,1] + 23.821;
   1:  PR[91,2] = PR[90,2] + 18.535;
   1:L PR[91] R[100]mm/sec CNT100;
   1:  PR[91,1] = PR[90,1] + 22.403;
   1:  PR[91,2] = PR[90,2] + 19.090;
   1:L PR[91] R[100]mm/sec CNT100;
   1:  PR[91,1] = PR[90,1] + 20.113;
   1:  PR[91,2] = PR[90,2] + 19.564;
   1:L PR[91] R[100]mm/sec CNT100;
   1:  PR[91,1] = PR[90,1] + 18.194;
   1:  PR[91,2] = PR[90,2] + 19.791;
   1:L PR[91] R[100]mm/sec CNT100;
   1:  PR[91,1] = PR[90,1] + 15.953;
   1:  PR[91,2] = PR[90,2] + 19.907;
   1:L PR[91] R[100]mm/sec CNT100;
   1:  PR[91,1] = PR[90,1] + 13.954;
   1:  PR[91,2] = PR[90,2] + 19.704;
   1:L PR[91] R[100]mm/sec CNT100;
   1:  PR[91,1] = PR[90,1] + 11.493;
   1:  PR[91,2] = PR[90,2] + 19.364;
   1:L PR[91] R[100]mm/sec CNT100;
   1:  PR[91,1] = PR[90,1] + 9.726;
   1:  PR[91,2] = PR[90,2] + 18.906;
   1:L PR[91] R[100]mm/sec CNT100;
   1:  PR[91,1] = PR[90,1] + 8.150;
   1:  PR[91,2] = PR[90,2] + 18.216;
   1:L PR[91] R[100]mm/sec CNT100;
   1:  PR[91,1] = PR[90,1] + 5.426;
   1:  PR[91,2] = PR[90,2] + 17.078;
   1:L PR[91] R[100]mm/sec CNT100;
   1:  PR[91,1] = PR[90,1] + 4.147;
   1:  PR[91,2] = PR[90,2] + 16.261;
   1:L PR[91] R[100]mm/sec CNT100;
   1:  PR[91,1] = PR[90,1] + 3.625;
   1:  PR[91,2] = PR[90,2] + 15.901;
   1:L PR[91] R[100]mm/sec CNT100;
   1:  PR[91,1] = PR[90,1] + 2.675;
   1:  PR[91,2] = PR[90,2] + 15.149;
   1:L PR[91] R[100]mm/sec CNT100;
   1:  PR[91,1] = PR[90,1] + 2.026;
   1:  PR[91,2] = PR[90,2] + 14.575;
   1:L PR[91] R[100]mm/sec CNT100;
   1:  PR[91,1] = PR[90,1] + 1.855;
   1:  PR[91,2] = PR[90,2] + 14.459;
   1:L PR[91] R[100]mm/sec CNT100;
   1:  PR[91,1] = PR[90,1] + 1.521;
   1:  PR[91,2] = PR[90,2] + 14.135;
   1:L PR[91] R[100]mm/sec CNT100;
   1:  PR[91,1] = PR[90,1] + 0.938;
   1:  PR[91,2] = PR[90,2] + 14.036;
   1:L PR[91] R[100]mm/sec CNT100;
   1:  PR[91,1] = PR[90,1] + 0.459;
   1:  PR[91,2] = PR[90,2] + 13.773;
   1:L PR[91] R[100]mm/sec CNT100;
   1:  PR[91,1] = PR[90,1] + -0.415;
   1:L PR[91] R[100]mm/sec CNT100;
   1:  PR[91] = PR[90];
   1:  PR[91,1] = PR[90,1] + -1.816;
   1:  PR[91,2] = PR[90,2] + 14.722;
   1:  PR[91,3] = PR[90,3] + 32.635;
   1:L PR[91] R[100]mm/sec CNT100;
   1:  PR[91,1] = PR[90,1] + -2.026;
   1:  PR[91,2] = PR[90,2] + 14.996;
   1:L PR[91] R[100]mm/sec CNT100;
   1:  PR[91,1] = PR[90,1] + -2.230;
   1:  PR[91,2] = PR[90,2] + 15.176;
   1:L PR[91] R[100]mm/sec CNT100;
   1:  PR[91,1] = PR[90,1] + -3.224;
   1:  PR[91,2] = PR[90,2] + 15.962;
   1:L PR[91] R[100]mm/sec CNT100;
   1:  PR[91,1] = PR[90,1] + -4.115;
   1:  PR[91,2] = PR[90,2] + 16.533;
   1:L PR[91] R[100]mm/sec CNT100;
   1:  PR[91,1] = PR[90,1] + -5.011;
   1:  PR[91,2] = PR[90,2] + 17.133;
   1:L PR[91] R[100]mm/sec CNT100;
   1:  PR[91,1] = PR[90,1] + -6.471;
   1:  PR[91,2] = PR[90,2] + 17.771;
   1:L PR[91] R[100]mm/sec CNT100;
   1:  PR[91,1] = PR[90,1] + -9.368;
   1:  PR[91,2] = PR[90,2] + 18.986;
   1:L PR[91] R[100]mm/sec CNT100;
   1:  PR[91,1] = PR[90,1] + -10.991;
   1:  PR[91,2] = PR[90,2] + 19.405;
   1:L PR[91] R[100]mm/sec CNT100;
   1:  PR[91,1] = PR[90,1] + -13.014;
   1:  PR[91,2] = PR[90,2] + 19.616;
   1:L PR[91] R[100]mm/sec CNT100;
   1:  PR[91,1] = PR[90,1] + -15.605;
   1:  PR[91,2] = PR[90,2] + 19.969;
   1:L PR[91] R[100]mm/sec CNT100;
   1:  PR[91,1] = PR[90,1] + -17.689;
   1:  PR[91,2] = PR[90,2] + 19.859;
   1:L PR[91] R[100]mm/sec CNT100;
   1:  PR[91,1] = PR[90,1] + -19.849;
   1:  PR[91,2] = PR[90,2] + 19.604;
   1:L PR[91] R[100]mm/sec CNT100;
   1:  PR[91,1] = PR[90,1] + -22.022;
   1:  PR[91,2] = PR[90,2] + 19.153;
   1:L PR[91] R[100]mm/sec CNT100;
   1:  PR[91,1] = PR[90,1] + -24.414;
   1:  PR[91,2] = PR[90,2] + 18.265;
   1:L PR[91] R[100]mm/sec CNT100;
   1:  PR[91,1] = PR[90,1] + -25.877;
   1:  PR[91,2] = PR[90,2] + 17.693;
   1:L PR[91] R[100]mm/sec CNT100;
   1:  PR[91,1] = PR[90,1] + -28.113;
   1:  PR[91,2] = PR[90,2] + 16.441;
   1:L PR[91] R[100]mm/sec CNT100;
   1:  PR[91,1] = PR[90,1] + -30.422;
   1:  PR[91,2] = PR[90,2] + 14.644;
   1:L PR[91] R[100]mm/sec CNT100;
   1:  PR[91,1] = PR[90,1] + -31.215;
   1:  PR[91,2] = PR[90,2] + 14.066;
   1:L PR[91] R[100]mm/sec CNT100;
   1:  PR[91,1] = PR[90,1] + -33.133;
   1:  PR[91,2] = PR[90,2] + 11.994;
   1:L PR[91] R[100]mm/sec CNT100;
   1:  PR[91,1] = PR[90,1] + -33.564;
   1:  PR[91,2] = PR[90,2] + 11.460;
   1:L PR[91] R[100]mm/sec CNT100;
   1:  PR[91,1] = PR[90,1] + -35.171;
   1:  PR[91,2] = PR[90,2] + 9.018;
   1:L PR[91] R[100]mm/sec CNT100;
   1:  PR[91,1] = PR[90,1] + -36.621;
   1:  PR[91,2] = PR[90,2] + 5.773;
   1:L PR[91] R[100]mm/sec CNT100;
   1:  PR[91,1] = PR[90,1] + -37.347;
   1:  PR[91,2] = PR[90,2] + 2.970;
   1:L PR[91] R[100]mm/sec CNT100;
   1:  PR[91,1] = PR[90,1] + -37.596;
   1:  PR[91,2] = PR[90,2] + -0.139;
   1:L PR[91] R[100]mm/sec CNT100;
   1:  PR[91,1] = PR[90,1] + -37.625;
   1:  PR[91,2] = PR[90,2] + -0.354;
   1:L PR[91] R[100]mm/sec CNT100;
   1:  PR[91,1] = PR[90,1] + -37.389;
   1:  PR[91,2] = PR[90,2] + -3.326;
   1:L PR[91] R[100]mm/sec CNT100;
   1:  PR[91,1] = PR[90,1] + -37.357;
   1:  PR[91,2] = PR[90,2] + -3.553;
   1:L PR[91] R[100]mm/sec CNT100;
   1:  PR[91,1] = PR[90,1] + -36.621;
   1:  PR[91,2] = PR[90,2] + -6.397;
   1:L PR[91] R[100]mm/sec CNT100;
   1:  PR[91,1] = PR[90,1] + -35.354;
   1:  PR[91,2] = PR[90,2] + -9.220;
   1:L PR[91] R[100]mm/sec CNT100;
   1:  PR[91,1] = PR[90,1] + -35.167;
   1:  PR[91,2] = PR[90,2] + -9.647;
   1:L PR[91] R[100]mm/sec CNT100;
   1:  PR[91,1] = PR[90,1] + -33.563;
   1:  PR[91,2] = PR[90,2] + -12.085;
   1:L PR[91] R[100]mm/sec CNT100;
   1:  PR[91,1] = PR[90,1] + -33.132;
   1:  PR[91,2] = PR[90,2] + -12.620;
   1:L PR[91] R[100]mm/sec CNT100;
   1:  PR[91,1] = PR[90,1] + -31.195;
   1:  PR[91,2] = PR[90,2] + -14.711;
   1:L PR[91] R[100]mm/sec CNT100;
   1:  PR[91,1] = PR[90,1] + -29.091;
   1:  PR[91,2] = PR[90,2] + -16.358;
   1:L PR[91] R[100]mm/sec CNT100;
   1:  PR[91,1] = PR[90,1] + -28.128;
   1:  PR[91,2] = PR[90,2] + -17.056;
   1:L PR[91] R[100]mm/sec CNT100;
   1:  PR[91,1] = PR[90,1] + -25.882;
   1:  PR[91,2] = PR[90,2] + -18.314;
   1:L PR[91] R[100]mm/sec CNT100;
   1:  PR[91,1] = PR[90,1] + -23.637;
   1:  PR[91,2] = PR[90,2] + -19.144;
   1:L PR[91] R[100]mm/sec CNT100;
   1:  PR[91,1] = PR[90,1] + -21.998;
   1:  PR[91,2] = PR[90,2] + -19.783;
   1:L PR[91] R[100]mm/sec CNT100;
   1:  PR[91,1] = PR[90,1] + -19.837;
   1:  PR[91,2] = PR[90,2] + -20.231;
   1:L PR[91] R[100]mm/sec CNT100;
   1:  PR[91,1] = PR[90,1] + -17.672;
   1:  PR[91,2] = PR[90,2] + -20.483;
   1:L PR[91] R[100]mm/sec CNT100;
   1:  PR[91,1] = PR[90,1] + -15.560;
   1:  PR[91,2] = PR[90,2] + -20.595;
   1:L PR[91] R[100]mm/sec CNT100;
   1:  PR[91,1] = PR[90,1] + -13.684;
   1:  PR[91,2] = PR[90,2] + -20.406;
   1:L PR[91] R[100]mm/sec CNT100;
   1:  PR[91,1] = PR[90,1] + -10.990;
   1:  PR[91,2] = PR[90,2] + -20.029;
   1:L PR[91] R[100]mm/sec CNT100;
   1:  PR[91,1] = PR[90,1] + -9.354;
   1:  PR[91,2] = PR[90,2] + -19.606;
   1:L PR[91] R[100]mm/sec CNT100;
   1:  PR[91,1] = PR[90,1] + -7.890;
   1:  PR[91,2] = PR[90,2] + -18.964;
   1:L PR[91] R[100]mm/sec CNT100;
   1:  PR[91,1] = PR[90,1] + -4.902;
   1:  PR[91,2] = PR[90,2] + -17.690;
   1:L PR[91] R[100]mm/sec CNT100;
   1:  PR[91,1] = PR[90,1] + -3.757;
   1:  PR[91,2] = PR[90,2] + -16.958;
   1:L PR[91] R[100]mm/sec CNT100;
   1:  PR[91,1] = PR[90,1] + -2.887;
   1:  PR[91,2] = PR[90,2] + -16.331;
   1:L PR[91] R[100]mm/sec CNT100;
   1:  PR[91,1] = PR[90,1] + -1.703;
   1:  PR[91,2] = PR[90,2] + -15.294;
   1:L PR[91] R[100]mm/sec CNT100;
   1:  PR[91,1] = PR[90,1] + -1.035;
   1:  PR[91,2] = PR[90,2] + -15.066;
   1:L PR[91] R[100]mm/sec CNT100;
   1:  PR[91,1] = PR[90,1] + -0.337;
   1:  PR[91,2] = PR[90,2] + -14.534;
   1:L PR[91] R[100]mm/sec CNT100;
   1:  PR[91,1] = PR[90,1] + 0.674;
   1:  PR[91,2] = PR[90,2] + -14.893;
   1:L PR[91] R[100]mm/sec CNT100;
   1:  PR[91,1] = PR[90,1] + 1.612;
   1:  PR[91,2] = PR[90,2] + -15.061;
   1:L PR[91] R[100]mm/sec CNT100;
   1:  PR[91,1] = PR[90,1] + 1.833;
   1:  PR[91,2] = PR[90,2] + -15.312;
   1:L PR[91] R[100]mm/sec CNT100;
   1:  PR[91,1] = PR[90,1] + 1.979;
   1:  PR[91,2] = PR[90,2] + -15.400;
   1:L PR[91] R[100]mm/sec CNT100;
   1:  PR[91,1] = PR[90,1] + 3.016;
   1:  PR[91,2] = PR[90,2] + -16.310;
   1:L PR[91] R[100]mm/sec CNT100;
   1:  PR[91,1] = PR[90,1] + 3.637;
   1:  PR[91,2] = PR[90,2] + -16.707;
   1:L PR[91] R[100]mm/sec CNT100;
   1:  PR[91,1] = PR[90,1] + 4.227;
   1:  PR[91,2] = PR[90,2] + -17.128;
   1:L PR[91] R[100]mm/sec CNT100;
   1:  PR[91,1] = PR[90,1] + 5.073;
   1:  PR[91,2] = PR[90,2] + -17.699;
   1:L PR[91] R[100]mm/sec CNT100;
   1:  PR[91,1] = PR[90,1] + 9.499;
   1:  PR[91,2] = PR[90,2] + -19.600;
   1:L PR[91] R[100]mm/sec CNT100;
   1:  PR[91,1] = PR[90,1] + 11.120;
   1:  PR[91,2] = PR[90,2] + -20.021;
   1:L PR[91] R[100]mm/sec CNT100;
   1:  PR[91,1] = PR[90,1] + 13.140;
   1:  PR[91,2] = PR[90,2] + -20.232;
   1:L PR[91] R[100]mm/sec CNT100;
   1:  PR[91,1] = PR[90,1] + 15.737;
   1:  PR[91,2] = PR[90,2] + -20.593;
   1:L PR[91] R[100]mm/sec CNT100;
   1:  PR[91,1] = PR[90,1] + 17.811;
   1:  PR[91,2] = PR[90,2] + -20.486;
   1:L PR[91] R[100]mm/sec CNT100;
   1:  PR[91,1] = PR[90,1] + 19.977;
   1:  PR[91,2] = PR[90,2] + -20.233;
   1:L PR[91] R[100]mm/sec CNT100;
   1:  PR[91,1] = PR[90,1] + 22.147;
   1:  PR[91,2] = PR[90,2] + -19.784;
   1:L PR[91] R[100]mm/sec CNT100;
   1:  PR[91,1] = PR[90,1] + 24.544;
   1:  PR[91,2] = PR[90,2] + -18.899;
   1:L PR[91] R[100]mm/sec CNT100;
   1:  PR[91,1] = PR[90,1] + 26.014;
   1:  PR[91,2] = PR[90,2] + -18.327;
   1:L PR[91] R[100]mm/sec CNT100;
   1:  PR[91,1] = PR[90,1] + 28.239;
   1:  PR[91,2] = PR[90,2] + -17.087;
   1:L PR[91] R[100]mm/sec CNT100;
   1:  PR[91,1] = PR[90,1] + 30.530;
   1:  PR[91,2] = PR[90,2] + -15.312;
   1:L PR[91] R[100]mm/sec CNT100;
   1:  PR[91,1] = PR[90,1] + 31.328;
   1:  PR[91,2] = PR[90,2] + -14.732;
   1:L PR[91] R[100]mm/sec CNT100;
   1:  PR[91,1] = PR[90,1] + 33.251;
   1:  PR[91,2] = PR[90,2] + -12.658;
   1:L PR[91] R[100]mm/sec CNT100;
   1:  PR[91,1] = PR[90,1] + 33.686;
   1:  PR[91,2] = PR[90,2] + -12.118;
   1:L PR[91] R[100]mm/sec CNT100;
   1:  PR[91,1] = PR[90,1] + 35.315;
   1:  PR[91,2] = PR[90,2] + -9.656;
   1:L PR[91] R[100]mm/sec CNT100;
   1:  PR[91,1] = PR[90,1] + 36.629;
   1:  PR[91,2] = PR[90,2] + -6.763;
   1:L PR[91] R[100]mm/sec CNT100;
   1:  PR[91,1] = PR[90,1] + 36.761;
   1:  PR[91,2] = PR[90,2] + -6.463;
   1:L PR[91] R[100]mm/sec CNT100;
   1:  PR[91,1] = PR[90,1] + 37.490;
   1:  PR[91,2] = PR[90,2] + -3.687;
   1:L PR[91] R[100]mm/sec CNT100;
   1:  PR[91,1] = PR[90,1] + 37.753;
   1:  PR[91,2] = PR[90,2] + -0.485;
   1:L PR[91] R[100]mm/sec CNT100;
   1:  PR[91,1] = PR[90,1] + 37.782;
   1:  PR[91,2] = PR[90,2] + -0.271;
